LIN {X 46.511,Y 61.150,Z 69.018,A 180.000,B 0.000,C 180.000} C_DIS
LIN {X 46.612,Y 61.449,Z 69.014,A 180.000,B 0.000,C 180.000} C_DIS
LIN {X 46.713,Y 61.747,Z 69.011,A 180.000,B 0.000,C 180.000} C_DIS
LIN {X 46.814,Y 62.046,Z 69.008,A 180.000,B 0.000,C 180.000} C_DIS
LIN {X 46.914,Y 62.344,Z 69.005,A 180.000,B 0.000,C 180.000} C_DIS
LIN {X 47.015,Y 62.643,Z 69.003,A 180.000,B 0.000,C 180.000} C_DIS
LIN {X 47.116,Y 62.941,Z 69.002,A 180.000,B 0.000,C 180.000} C_DIS
LIN {X 47.216,Y 63.240,Z 69.001,A 180.000,B 0.000,C 180.000} C_DIS
LIN {X 47.317,Y 63.538,Z 69.000,A 180.000,B 0.000,C 180.000} C_DIS
LIN {X 47.391,Y 63.759,Z 69.000,A 180.000,B 0.000,C 180.000} C_DIS
; Cutting Move Starts
LIN {X 50.248,Y 72.226,Z 69.000,A 180.000,B 0.000,C 180.000} C_DIS
LIN {X 50.311,Y 72.405,Z 69.000,A 180.000,B 0.000,C 180.000} C_DIS
LIN {X 50.388,Y 72.584,Z 69.000,A 180.000,B 0.000,C 180.000} C_DIS
LIN {X 50.416,Y 72.640,Z 69.000,A 180.000,B 0.000,C 180.000} C_DIS
LIN {X 50.484,Y 72.763,Z 69.000,A 180.000,B 0.000,C 180.000} C_DIS
LIN {X 50.595,Y 72.936,Z 69.000,A 180.000,B 0.000,C 180.000} C_DIS
LIN {X 50.599,Y 72.941,Z 69.000,A 180.000,B 0.000,C 180.000} C_DIS
LIN {X 50.665,Y 73.031,Z 69.000,A 180.000,B 0.000,C 180.000} C_DIS
LIN {X 50.737,Y 73.120,Z 69.000,A 180.000,B 0.000,C 180.000} C_DIS
LIN {X 50.774,Y 73.162,Z 69.000,A 180.000,B 0.000,C 180.000} C_DIS
LIN {X 50.905,Y 73.299,Z 69.000,A 180.000,B 0.000,C 180.000} C_DIS
LIN {X 50.953,Y 73.343,Z 69.000,A 180.000,B 0.000,C 180.000} C_DIS
LIN {X 51.112,Y 73.478,Z 69.000,A 180.000,B 0.000,C 180.000} C_DIS
LIN {X 51.131,Y 73.493,Z 69.000,A 180.000,B 0.000,C 180.000} C_DIS
LIN {X 51.310,Y 73.616,Z 69.000,A 180.000,B 0.000,C 180.000} C_DIS
LIN {X 51.376,Y 73.656,Z 69.000,A 180.000,B 0.000,C 180.000} C_DIS
LIN {X 51.489,Y 73.719,Z 69.000,A 180.000,B 0.000,C 180.000} C_DIS
LIN {X 51.668,Y 73.803,Z 69.000,A 180.000,B 0.000,C 180.000} C_DIS
LIN {X 51.749,Y 73.835,Z 69.000,A 180.000,B 0.000,C 180.000} C_DIS
LIN {X 51.847,Y 73.870,Z 69.000,A 180.000,B 0.000,C 180.000} C_DIS
LIN {X 52.025,Y 73.923,Z 69.000,A 180.000,B 0.000,C 180.000} C_DIS
LIN {X 52.204,Y 73.961,Z 69.000,A 180.000,B 0.000,C 180.000} C_DIS
LIN {X 52.383,Y 73.987,Z 69.000,A 180.000,B 0.000,C 180.000} C_DIS
LIN {X 52.562,Y 73.999,Z 69.000,A 180.000,B 0.000,C 180.000} C_DIS
LIN {X 52.740,Y 73.998,Z 69.000,A 180.000,B 0.000,C 180.000} C_DIS
LIN {X 52.919,Y 73.985,Z 69.000,A 180.000,B 0.000,C 180.000} C_DIS
LIN {X 53.098,Y 73.958,Z 69.000,A 180.000,B 0.000,C 180.000} C_DIS
LIN {X 53.277,Y 73.918,Z 69.000,A 180.000,B 0.000,C 180.000} C_DIS
LIN {X 53.455,Y 73.864,Z 69.000,A 180.000,B 0.000,C 180.000} C_DIS
LIN {X 83.198,Y 63.830,Z 69.000,A 180.000,B 0.000,C 180.000} C_DIS
LIN {X 96.464,Y 59.355,Z 69.000,A 180.000,B 0.000,C 180.000} C_DIS
LIN {X 96.539,Y 59.329,Z 69.000,A 180.000,B 0.000,C 180.000} C_DIS
LIN {X 96.718,Y 59.257,Z 69.000,A 180.000,B 0.000,C 180.000} C_DIS
LIN {X 96.883,Y 59.176,Z 69.000,A 180.000,B 0.000,C 180.000} C_DIS
LIN {X 96.897,Y 59.169,Z 69.000,A 180.000,B 0.000,C 180.000} C_DIS
LIN {X 97.075,Y 59.061,Z 69.000,A 180.000,B 0.000,C 180.000} C_DIS
LIN {X 97.167,Y 58.997,Z 69.000,A 180.000,B 0.000,C 180.000} C_DIS
LIN {X 97.254,Y 58.931,Z 69.000,A 180.000,B 0.000,C 180.000} C_DIS
LIN {X 97.385,Y 58.819,Z 69.000,A 180.000,B 0.000,C 180.000} C_DIS
LIN {X 97.433,Y 58.774,Z 69.000,A 180.000,B 0.000,C 180.000} C_DIS
LIN {X 97.562,Y 58.640,Z 69.000,A 180.000,B 0.000,C 180.000} C_DIS
LIN {X 97.612,Y 58.582,Z 69.000,A 180.000,B 0.000,C 180.000} C_DIS
LIN {X 97.707,Y 58.461,Z 69.000,A 180.000,B 0.000,C 180.000} C_DIS
LIN {X 97.790,Y 58.341,Z 69.000,A 180.000,B 0.000,C 180.000} C_DIS
LIN {X 97.828,Y 58.282,Z 69.000,A 180.000,B 0.000,C 180.000} C_DIS
LIN {X 97.928,Y 58.103,Z 69.000,A 180.000,B 0.000,C 180.000} C_DIS
LIN {X 97.969,Y 58.017,Z 69.000,A 180.000,B 0.000,C 180.000} C_DIS
LIN {X 98.009,Y 57.925,Z 69.000,A 180.000,B 0.000,C 180.000} C_DIS
LIN {X 98.075,Y 57.746,Z 69.000,A 180.000,B 0.000,C 180.000} C_DIS
LIN {X 98.125,Y 57.567,Z 69.000,A 180.000,B 0.000,C 180.000} C_DIS
LIN {X 98.148,Y 57.466,Z 69.000,A 180.000,B 0.000,C 180.000} C_DIS
LIN {X 98.162,Y 57.388,Z 69.000,A 180.000,B 0.000,C 180.000} C_DIS
LIN {X 98.186,Y 57.210,Z 69.000,A 180.000,B 0.000,C 180.000} C_DIS
LIN {X 98.196,Y 57.031,Z 69.000,A 180.000,B 0.000,C 180.000} C_DIS
LIN {X 98.193,Y 56.852,Z 69.000,A 180.000,B 0.000,C 180.000} C_DIS
LIN {X 98.178,Y 56.673,Z 69.000,A 180.000,B 0.000,C 180.000} C_DIS
LIN {X 98.150,Y 56.495,Z 69.000,A 180.000,B 0.000,C 180.000} C_DIS
LIN {X 98.148,Y 56.485,Z 69.000,A 180.000,B 0.000,C 180.000} C_DIS
LIN {X 98.108,Y 56.316,Z 69.000,A 180.000,B 0.000,C 180.000} C_DIS
LIN {X 98.052,Y 56.137,Z 69.000,A 180.000,B 0.000,C 180.000} C_DIS
LIN {X 97.793,Y 55.369,Z 69.000,A 180.000,B 0.000,C 180.000} C_DIS
LIN {X 97.793,Y 55.367,Z 69.000,A 180.000,B 0.000,C 180.000} C_DIS
LIN {X 97.971,Y 55.243,Z 69.000,A 180.000,B 0.000,C 180.000} C_DIS
LIN {X 98.148,Y 55.119,Z 69.000,A 180.000,B 0.000,C 180.000} C_DIS
LIN {X 98.220,Y 55.064,Z 69.000,A 180.000,B 0.000,C 180.000} C_DIS
LIN {X 98.505,Y 54.838,Z 69.000,A 180.000,B 0.000,C 180.000} C_DIS
LIN {X 98.665,Y 54.707,Z 69.000,A 180.000,B 0.000,C 180.000} C_DIS
LIN {X 98.684,Y 54.690,Z 69.000,A 180.000,B 0.000,C 180.000} C_DIS
LIN {X 98.863,Y 54.528,Z 69.000,A 180.000,B 0.000,C 180.000} C_DIS
LIN {X 99.042,Y 54.367,Z 69.000,A 180.000,B 0.000,C 180.000} C_DIS
LIN {X 99.060,Y 54.349,Z 69.000,A 180.000,B 0.000,C 180.000} C_DIS
LIN {X 99.221,Y 54.188,Z 69.000,A 180.000,B 0.000,C 180.000} C_DIS
LIN {X 99.412,Y 53.992,Z 69.000,A 180.000,B 0.000,C 180.000} C_DIS
LIN {X 99.575,Y 53.813,Z 69.000,A 180.000,B 0.000,C 180.000} C_DIS
LIN {X 99.757,Y 53.602,Z 69.000,A 180.000,B 0.000,C 180.000} C_DIS
LIN {X 99.881,Y 53.455,Z 69.000,A 180.000,B 0.000,C 180.000} C_DIS
LIN {X 99.936,Y 53.385,Z 69.000,A 180.000,B 0.000,C 180.000} C_DIS
LIN {X 100.153,Y 53.098,Z 69.000,A 180.000,B 0.000,C 180.000} C_DIS
LIN {X 100.282,Y 52.919,Z 69.000,A 180.000,B 0.000,C 180.000} C_DIS
LIN {X 100.520,Y 52.562,Z 69.000,A 180.000,B 0.000,C 180.000} C_DIS
LIN {X 100.629,Y 52.383,Z 69.000,A 180.000,B 0.000,C 180.000} C_DIS
LIN {X 100.732,Y 52.204,Z 69.000,A 180.000,B 0.000,C 180.000} C_DIS
LIN {X 100.829,Y 52.034,Z 69.000,A 180.000,B 0.000,C 180.000} C_DIS
LIN {X 100.835,Y 52.025,Z 69.000,A 180.000,B 0.000,C 180.000} C_DIS
LIN {X 100.927,Y 51.847,Z 69.000,A 180.000,B 0.000,C 180.000} C_DIS
LIN {X 101.016,Y 51.668,Z 69.000,A 180.000,B 0.000,C 180.000} C_DIS
LIN {X 101.104,Y 51.489,Z 69.000,A 180.000,B 0.000,C 180.000} C_DIS
LIN {X 101.183,Y 51.310,Z 69.000,A 180.000,B 0.000,C 180.000} C_DIS
LIN {X 101.258,Y 51.131,Z 69.000,A 180.000,B 0.000,C 180.000} C_DIS
LIN {X 101.333,Y 50.953,Z 69.000,A 180.000,B 0.000,C 180.000} C_DIS
LIN {X 101.366,Y 50.869,Z 69.000,A 180.000,B 0.000,C 180.000} C_DIS
LIN {X 101.399,Y 50.774,Z 69.000,A 180.000,B 0.000,C 180.000} C_DIS
LIN {X 101.523,Y 50.416,Z 69.000,A 180.000,B 0.000,C 180.000} C_DIS
LIN {X 101.545,Y 50.354,Z 69.000,A 180.000,B 0.000,C 180.000} C_DIS
LIN {X 101.579,Y 50.238,Z 69.000,A 180.000,B 0.000,C 180.000} C_DIS
LIN {X 101.679,Y 49.880,Z 69.000,A 180.000,B 0.000,C 180.000} C_DIS
LIN {X 101.723,Y 49.708,Z 69.000,A 180.000,B 0.000,C 180.000} C_DIS
LIN {X 101.725,Y 49.701,Z 69.000,A 180.000,B 0.000,C 180.000} C_DIS
LIN {X 101.763,Y 49.523,Z 69.000,A 180.000,B 0.000,C 180.000} C_DIS
LIN {X 101.801,Y 49.344,Z 69.000,A 180.000,B 0.000,C 180.000} C_DIS
LIN {X 101.837,Y 49.165,Z 69.000,A 180.000,B 0.000,C 180.000} C_DIS
LIN {X 101.864,Y 48.986,Z 69.000,A 180.000,B 0.000,C 180.000} C_DIS
LIN {X 101.902,Y 48.729,Z 69.000,A 180.000,B 0.000,C 180.000} C_DIS
LIN {X 101.917,Y 48.629,Z 69.000,A 180.000,B 0.000,C 180.000} C_DIS
LIN {X 101.935,Y 48.450,Z 69.000,A 180.000,B 0.000,C 180.000} C_DIS
LIN {X 101.964,Y 48.092,Z 69.000,A 180.000,B 0.000,C 180.000} C_DIS
LIN {X 101.974,Y 47.914,Z 69.000,A 180.000,B 0.000,C 180.000} C_DIS
LIN {X 101.982,Y 47.556,Z 69.000,A 180.000,B 0.000,C 180.000} C_DIS
LIN {X 101.983,Y 47.377,Z 69.000,A 180.000,B 0.000,C 180.000} C_DIS
LIN {X 101.977,Y 47.198,Z 69.000,A 180.000,B 0.000,C 180.000} C_DIS
LIN {X 101.969,Y 47.020,Z 69.000,A 180.000,B 0.000,C 180.000} C_DIS
LIN {X 101.961,Y 46.841,Z 69.000,A 180.000,B 0.000,C 180.000} C_DIS
LIN {X 101.945,Y 46.662,Z 69.000,A 180.000,B 0.000,C 180.000} C_DIS
LIN {X 101.907,Y 46.305,Z 69.000,A 180.000,B 0.000,C 180.000} C_DIS
LIN {X 101.902,Y 46.257,Z 69.000,A 180.000,B 0.000,C 180.000} C_DIS
LIN {X 101.883,Y 46.126,Z 69.000,A 180.000,B 0.000,C 180.000} C_DIS
LIN {X 101.822,Y 45.768,Z 69.000,A 180.000,B 0.000,C 180.000} C_DIS
LIN {X 101.790,Y 45.590,Z 69.000,A 180.000,B 0.000,C 180.000} C_DIS
LIN {X 101.748,Y 45.411,Z 69.000,A 180.000,B 0.000,C 180.000} C_DIS
LIN {X 101.706,Y 45.232,Z 69.000,A 180.000,B 0.000,C 180.000} C_DIS
LIN {X 101.663,Y 45.053,Z 69.000,A 180.000,B 0.000,C 180.000} C_DIS
LIN {X 101.611,Y 44.874,Z 69.000,A 180.000,B 0.000,C 180.000} C_DIS
LIN {X 101.545,Y 44.655,Z 69.000,A 180.000,B 0.000,C 180.000} C_DIS
LIN {X 101.503,Y 44.517,Z 69.000,A 180.000,B 0.000,C 180.000} C_DIS
LIN {X 101.439,Y 44.338,Z 69.000,A 180.000,B 0.000,C 180.000} C_DIS
LIN {X 101.306,Y 43.981,Z 69.000,A 180.000,B 0.000,C 180.000} C_DIS
LIN {X 101.232,Y 43.802,Z 69.000,A 180.000,B 0.000,C 180.000} C_DIS
LIN {X 101.072,Y 43.444,Z 69.000,A 180.000,B 0.000,C 180.000} C_DIS
LIN {X 101.008,Y 43.311,Z 69.000,A 180.000,B 0.000,C 180.000} C_DIS
LIN {X 100.985,Y 43.266,Z 69.000,A 180.000,B 0.000,C 180.000} C_DIS
LIN {X 100.797,Y 42.908,Z 69.000,A 180.000,B 0.000,C 180.000} C_DIS
LIN {X 100.695,Y 42.729,Z 69.000,A 180.000,B 0.000,C 180.000} C_DIS
LIN {X 100.586,Y 42.550,Z 69.000,A 180.000,B 0.000,C 180.000} C_DIS
LIN {X 100.478,Y 42.372,Z 69.000,A 180.000,B 0.000,C 180.000} C_DIS
LIN {X 100.472,Y 42.362,Z 69.000,A 180.000,B 0.000,C 180.000} C_DIS
LIN {X 100.357,Y 42.193,Z 69.000,A 180.000,B 0.000,C 180.000} C_DIS
LIN {X 100.233,Y 42.014,Z 69.000,A 180.000,B 0.000,C 180.000} C_DIS
LIN {X 100.114,Y 41.846,Z 69.000,A 180.000,B 0.000,C 180.000} C_DIS
LIN {X 100.107,Y 41.835,Z 69.000,A 180.000,B 0.000,C 180.000} C_DIS
LIN {X 99.966,Y 41.657,Z 69.000,A 180.000,B 0.000,C 180.000} C_DIS
LIN {X 99.824,Y 41.478,Z 69.000,A 180.000,B 0.000,C 180.000} C_DIS
LIN {X 99.757,Y 41.394,Z 69.000,A 180.000,B 0.000,C 180.000} C_DIS
LIN {X 99.675,Y 41.299,Z 69.000,A 180.000,B 0.000,C 180.000} C_DIS
LIN {X 99.399,Y 40.994,Z 69.000,A 180.000,B 0.000,C 180.000} C_DIS
LIN {X 99.351,Y 40.942,Z 69.000,A 180.000,B 0.000,C 180.000} C_DIS
LIN {X 99.221,Y 40.811,Z 69.000,A 180.000,B 0.000,C 180.000} C_DIS
LIN {X 98.988,Y 40.584,Z 69.000,A 180.000,B 0.000,C 180.000} C_DIS
LIN {X 98.863,Y 40.468,Z 69.000,A 180.000,B 0.000,C 180.000} C_DIS
LIN {X 98.790,Y 40.405,Z 69.000,A 180.000,B 0.000,C 180.000} C_DIS
LIN {X 98.583,Y 40.226,Z 69.000,A 180.000,B 0.000,C 180.000} C_DIS
LIN {X 98.505,Y 40.160,Z 69.000,A 180.000,B 0.000,C 180.000} C_DIS
LIN {X 98.363,Y 40.048,Z 69.000,A 180.000,B 0.000,C 180.000} C_DIS
LIN {X 98.127,Y 39.869,Z 69.000,A 180.000,B 0.000,C 180.000} C_DIS
LIN {X 97.969,Y 39.752,Z 69.000,A 180.000,B 0.000,C 180.000} C_DIS
LIN {X 97.878,Y 39.690,Z 69.000,A 180.000,B 0.000,C 180.000} C_DIS
LIN {X 97.608,Y 39.511,Z 69.000,A 180.000,B 0.000,C 180.000} C_DIS
LIN {X 97.433,Y 39.400,Z 69.000,A 180.000,B 0.000,C 180.000} C_DIS
LIN {X 97.315,Y 39.333,Z 69.000,A 180.000,B 0.000,C 180.000} C_DIS
LIN {X 97.075,Y 39.194,Z 69.000,A 180.000,B 0.000,C 180.000} C_DIS
LIN {X 97.004,Y 39.154,Z 69.000,A 180.000,B 0.000,C 180.000} C_DIS
LIN {X 96.897,Y 39.098,Z 69.000,A 180.000,B 0.000,C 180.000} C_DIS
LIN {X 96.539,Y 38.920,Z 69.000,A 180.000,B 0.000,C 180.000} C_DIS
LIN {X 96.360,Y 38.838,Z 69.000,A 180.000,B 0.000,C 180.000} C_DIS
LIN {X 96.003,Y 38.688,Z 69.000,A 180.000,B 0.000,C 180.000} C_DIS
LIN {X 95.824,Y 38.618,Z 69.000,A 180.000,B 0.000,C 180.000} C_DIS
LIN {X 95.466,Y 38.494,Z 69.000,A 180.000,B 0.000,C 180.000} C_DIS
LIN {X 95.301,Y 38.439,Z 69.000,A 180.000,B 0.000,C 180.000} C_DIS
LIN {X 95.288,Y 38.435,Z 69.000,A 180.000,B 0.000,C 180.000} C_DIS
LIN {X 95.109,Y 38.385,Z 69.000,A 180.000,B 0.000,C 180.000} C_DIS
LIN {X 94.930,Y 38.335,Z 69.000,A 180.000,B 0.000,C 180.000} C_DIS
LIN {X 94.751,Y 38.287,Z 69.000,A 180.000,B 0.000,C 180.000} C_DIS
LIN {X 94.630,Y 38.260,Z 69.000,A 180.000,B 0.000,C 180.000} C_DIS
LIN {X 94.394,Y 38.210,Z 69.000,A 180.000,B 0.000,C 180.000} C_DIS
LIN {X 94.215,Y 38.172,Z 69.000,A 180.000,B 0.000,C 180.000} C_DIS
LIN {X 94.036,Y 38.143,Z 69.000,A 180.000,B 0.000,C 180.000} C_DIS
LIN {X 93.679,Y 38.091,Z 69.000,A 180.000,B 0.000,C 180.000} C_DIS
LIN {X 93.612,Y 38.081,Z 69.000,A 180.000,B 0.000,C 180.000} C_DIS
LIN {X 93.500,Y 38.070,Z 69.000,A 180.000,B 0.000,C 180.000} C_DIS
LIN {X 93.142,Y 38.040,Z 69.000,A 180.000,B 0.000,C 180.000} C_DIS
LIN {X 92.964,Y 38.027,Z 69.000,A 180.000,B 0.000,C 180.000} C_DIS
LIN {X 92.785,Y 38.023,Z 69.000,A 180.000,B 0.000,C 180.000} C_DIS
LIN {X 92.606,Y 38.019,Z 69.000,A 180.000,B 0.000,C 180.000} C_DIS
LIN {X 92.427,Y 38.016,Z 69.000,A 180.000,B 0.000,C 180.000} C_DIS
LIN {X 92.249,Y 38.021,Z 69.000,A 180.000,B 0.000,C 180.000} C_DIS
LIN {X 91.946,Y 38.034,Z 69.000,A 180.000,B 0.000,C 180.000} C_DIS
LIN {X 91.944,Y 38.032,Z 69.000,A 180.000,B 0.000,C 180.000} C_DIS
LIN {X 91.712,Y 37.344,Z 69.000,A 180.000,B 0.000,C 180.000} C_DIS
LIN {X 91.659,Y 37.187,Z 69.000,A 180.000,B 0.000,C 180.000} C_DIS
LIN {X 91.588,Y 37.009,Z 69.000,A 180.000,B 0.000,C 180.000} C_DIS
LIN {X 91.533,Y 36.894,Z 69.000,A 180.000,B 0.000,C 180.000} C_DIS
LIN {X 91.500,Y 36.830,Z 69.000,A 180.000,B 0.000,C 180.000} C_DIS
LIN {X 91.392,Y 36.651,Z 69.000,A 180.000,B 0.000,C 180.000} C_DIS
LIN {X 91.355,Y 36.595,Z 69.000,A 180.000,B 0.000,C 180.000} C_DIS
LIN {X 91.263,Y 36.472,Z 69.000,A 180.000,B 0.000,C 180.000} C_DIS
LIN {X 91.176,Y 36.368,Z 69.000,A 180.000,B 0.000,C 180.000} C_DIS
LIN {X 91.107,Y 36.294,Z 69.000,A 180.000,B 0.000,C 180.000} C_DIS
LIN {X 90.997,Y 36.186,Z 69.000,A 180.000,B 0.000,C 180.000} C_DIS
LIN {X 90.917,Y 36.115,Z 69.000,A 180.000,B 0.000,C 180.000} C_DIS
LIN {X 90.818,Y 36.036,Z 69.000,A 180.000,B 0.000,C 180.000} C_DIS
LIN {X 90.677,Y 35.936,Z 69.000,A 180.000,B 0.000,C 180.000} C_DIS
LIN {X 90.640,Y 35.912,Z 69.000,A 180.000,B 0.000,C 180.000} C_DIS
LIN {X 90.461,Y 35.809,Z 69.000,A 180.000,B 0.000,C 180.000} C_DIS
LIN {X 90.356,Y 35.757,Z 69.000,A 180.000,B 0.000,C 180.000} C_DIS
LIN {X 90.282,Y 35.724,Z 69.000,A 180.000,B 0.000,C 180.000} C_DIS
LIN {X 90.103,Y 35.656,Z 69.000,A 180.000,B 0.000,C 180.000} C_DIS
LIN {X 89.925,Y 35.603,Z 69.000,A 180.000,B 0.000,C 180.000} C_DIS
LIN {X 89.819,Y 35.578,Z 69.000,A 180.000,B 0.000,C 180.000} C_DIS
LIN {X 89.746,Y 35.564,Z 69.000,A 180.000,B 0.000,C 180.000} C_DIS
LIN {X 89.567,Y 35.539,Z 69.000,A 180.000,B 0.000,C 180.000} C_DIS
LIN {X 89.388,Y 35.526,Z 69.000,A 180.000,B 0.000,C 180.000} C_DIS
LIN {X 89.209,Y 35.526,Z 69.000,A 180.000,B 0.000,C 180.000} C_DIS
LIN {X 89.031,Y 35.540,Z 69.000,A 180.000,B 0.000,C 180.000} C_DIS
LIN {X 88.852,Y 35.566,Z 69.000,A 180.000,B 0.000,C 180.000} C_DIS
LIN {X 88.788,Y 35.578,Z 69.000,A 180.000,B 0.000,C 180.000} C_DIS
LIN {X 88.673,Y 35.605,Z 69.000,A 180.000,B 0.000,C 180.000} C_DIS
LIN {X 88.494,Y 35.659,Z 69.000,A 180.000,B 0.000,C 180.000} C_DIS
LIN {X 66.460,Y 43.092,Z 69.000,A 180.000,B 0.000,C 180.000} C_DIS
LIN {X 45.590,Y 50.133,Z 69.000,A 180.000,B 0.000,C 180.000} C_DIS
LIN {X 45.411,Y 50.194,Z 69.000,A 180.000,B 0.000,C 180.000} C_DIS
LIN {X 45.296,Y 50.238,Z 69.000,A 180.000,B 0.000,C 180.000} C_DIS
LIN {X 45.232,Y 50.265,Z 69.000,A 180.000,B 0.000,C 180.000} C_DIS
LIN {X 45.053,Y 50.353,Z 69.000,A 180.000,B 0.000,C 180.000} C_DIS
LIN {X 44.944,Y 50.416,Z 69.000,A 180.000,B 0.000,C 180.000} C_DIS
LIN {X 44.874,Y 50.461,Z 69.000,A 180.000,B 0.000,C 180.000} C_DIS
LIN {X 44.785,Y 50.522,Z 69.000,A 180.000,B 0.000,C 180.000} C_DIS
LIN {X 44.696,Y 50.590,Z 69.000,A 180.000,B 0.000,C 180.000} C_DIS
LIN {X 44.689,Y 50.595,Z 69.000,A 180.000,B 0.000,C 180.000} C_DIS
LIN {X 44.603,Y 50.667,Z 69.000,A 180.000,B 0.000,C 180.000} C_DIS
LIN {X 44.517,Y 50.746,Z 69.000,A 180.000,B 0.000,C 180.000} C_DIS
LIN {X 44.488,Y 50.774,Z 69.000,A 180.000,B 0.000,C 180.000} C_DIS
LIN {X 44.410,Y 50.855,Z 69.000,A 180.000,B 0.000,C 180.000} C_DIS
LIN {X 44.338,Y 50.936,Z 69.000,A 180.000,B 0.000,C 180.000} C_DIS
LIN {X 44.325,Y 50.953,Z 69.000,A 180.000,B 0.000,C 180.000} C_DIS
LIN {X 44.254,Y 51.042,Z 69.000,A 180.000,B 0.000,C 180.000} C_DIS
LIN {X 44.189,Y 51.131,Z 69.000,A 180.000,B 0.000,C 180.000} C_DIS
LIN {X 44.159,Y 51.176,Z 69.000,A 180.000,B 0.000,C 180.000} C_DIS
LIN {X 44.077,Y 51.310,Z 69.000,A 180.000,B 0.000,C 180.000} C_DIS
LIN {X 43.984,Y 51.489,Z 69.000,A 180.000,B 0.000,C 180.000} C_DIS
LIN {X 43.981,Y 51.497,Z 69.000,A 180.000,B 0.000,C 180.000} C_DIS
LIN {X 43.909,Y 51.668,Z 69.000,A 180.000,B 0.000,C 180.000} C_DIS
LIN {X 43.849,Y 51.847,Z 69.000,A 180.000,B 0.000,C 180.000} C_DIS
LIN {X 43.804,Y 52.025,Z 69.000,A 180.000,B 0.000,C 180.000} C_DIS
LIN {X 43.802,Y 52.035,Z 69.000,A 180.000,B 0.000,C 180.000} C_DIS
LIN {X 43.772,Y 52.204,Z 69.000,A 180.000,B 0.000,C 180.000} C_DIS
LIN {X 43.754,Y 52.383,Z 69.000,A 180.000,B 0.000,C 180.000} C_DIS
LIN {X 43.748,Y 52.562,Z 69.000,A 180.000,B 0.000,C 180.000} C_DIS
LIN {X 43.756,Y 52.740,Z 69.000,A 180.000,B 0.000,C 180.000} C_DIS
LIN {X 43.776,Y 52.919,Z 69.000,A 180.000,B 0.000,C 180.000} C_DIS
LIN {X 43.802,Y 53.064,Z 69.000,A 180.000,B 0.000,C 180.000} C_DIS
LIN {X 43.809,Y 53.098,Z 69.000,A 180.000,B 0.000,C 180.000} C_DIS
LIN {X 43.856,Y 53.277,Z 69.000,A 180.000,B 0.000,C 180.000} C_DIS
LIN {X 43.916,Y 53.455,Z 69.000,A 180.000,B 0.000,C 180.000} C_DIS
LIN {X 47.391,Y 63.759,Z 69.000,A 180.000,B 0.000,C 180.000} C_DIS
; Link Move Starts
LIN {X 47.492,Y 64.057,Z 69.000,A 180.000,B 0.000,C 180.000} C_DIS
LIN {X 47.593,Y 64.356,Z 68.999,A 180.000,B 0.000,C 180.000} C_DIS
LIN {X 47.693,Y 64.654,Z 68.998,A 180.000,B 0.000,C 180.000} C_DIS
LIN {X 47.794,Y 64.953,Z 68.996,A 180.000,B 0.000,C 180.000} C_DIS
LIN {X 47.895,Y 65.251,Z 68.994,A 180.000,B 0.000,C 180.000} C_DIS
LIN {X 47.996,Y 65.550,Z 68.991,A 180.000,B 0.000,C 180.000} C_DIS
LIN {X 48.096,Y 65.848,Z 68.988,A 180.000,B 0.000,C 180.000} C_DIS
LIN {X 48.197,Y 66.147,Z 68.985,A 180.000,B 0.000,C 180.000} C_DIS
LIN {X 48.298,Y 66.445,Z 68.981,A 180.000,B 0.000,C 180.000} C_DIS
LIN {X 48.398,Y 66.743,Z 68.977,A 180.000,B 0.000,C 180.000} C_DIS
LIN {X 48.499,Y 67.042,Z 68.972,A 180.000,B 0.000,C 180.000} C_DIS
LIN {X 48.549,Y 67.191,Z 68.969,A 180.000,B 0.000,C 180.000} C_DIS
LIN {X 48.600,Y 67.340,Z 68.967,A 180.000,B 0.000,C 180.000} C_DIS
LIN {X 48.650,Y 67.490,Z 68.964,A 180.000,B 0.000,C 180.000} C_DIS
LIN {X 48.700,Y 67.639,Z 68.961,A 180.000,B 0.000,C 180.000} C_DIS
LIN {X 48.751,Y 67.788,Z 68.959,A 180.000,B 0.000,C 180.000} C_DIS
LIN {X 48.801,Y 67.937,Z 68.956,A 180.000,B 0.000,C 180.000} C_DIS
LIN {X 48.851,Y 68.087,Z 68.952,A 180.000,B 0.000,C 180.000} C_DIS
LIN {X 48.902,Y 68.236,Z 68.949,A 180.000,B 0.000,C 180.000} C_DIS
LIN {X 48.952,Y 68.385,Z 68.946,A 180.000,B 0.000,C 180.000} C_DIS
LIN {X 49.002,Y 68.534,Z 68.943,A 180.000,B 0.000,C 180.000} C_DIS
LIN {X 49.053,Y 68.684,Z 68.939,A 180.000,B 0.000,C 180.000} C_DIS
LIN {X 49.103,Y 68.833,Z 68.936,A 180.000,B 0.000,C 180.000} C_DIS
LIN {X 49.153,Y 68.982,Z 68.932,A 180.000,B 0.000,C 180.000} C_DIS
LIN {X 49.204,Y 69.131,Z 68.928,A 180.000,B 0.000,C 180.000} C_DIS
LIN {X 49.254,Y 69.280,Z 68.925,A 180.000,B 0.000,C 180.000} C_DIS
LIN {X 49.304,Y 69.430,Z 68.921,A 180.000,B 0.000,C 180.000} C_DIS
LIN {X 49.355,Y 69.579,Z 68.917,A 180.000,B 0.000,C 180.000} C_DIS
LIN {X 49.405,Y 69.728,Z 68.913,A 180.000,B 0.000,C 180.000} C_DIS
LIN {X 49.456,Y 69.877,Z 68.909,A 180.000,B 0.000,C 180.000} C_DIS
LIN {X 49.506,Y 70.027,Z 68.905,A 180.000,B 0.000,C 180.000} C_DIS
LIN {X 49.556,Y 70.176,Z 68.900,A 180.000,B 0.000,C 180.000} C_DIS
LIN {X 49.607,Y 70.325,Z 68.896,A 180.000,B 0.000,C 180.000} C_DIS
LIN {X 49.657,Y 70.474,Z 68.892,A 180.000,B 0.000,C 180.000} C_DIS
LIN {X 49.707,Y 70.624,Z 68.887,A 180.000,B 0.000,C 180.000} C_DIS
LIN {X 49.758,Y 70.773,Z 68.883,A 180.000,B 0.000,C 180.000} C_DIS
LIN {X 49.808,Y 70.922,Z 68.878,A 180.000,B 0.000,C 180.000} C_DIS
LIN {X 49.858,Y 71.071,Z 68.873,A 180.000,B 0.000,C 180.000} C_DIS
LIN {X 49.909,Y 71.221,Z 68.869,A 180.000,B 0.000,C 180.000} C_DIS
LIN {X 49.959,Y 71.370,Z 68.864,A 180.000,B 0.000,C 180.000} C_DIS
LIN {X 50.009,Y 71.519,Z 68.859,A 180.000,B 0.000,C 180.000} C_DIS
LIN {X 50.060,Y 71.668,Z 68.854,A 180.000,B 0.000,C 180.000} C_DIS
LIN {X 50.085,Y 71.743,Z 68.851,A 180.000,B 0.000,C 180.000} C_DIS
LIN {X 50.110,Y 71.818,Z 68.849,A 180.000,B 0.000,C 180.000} C_DIS
LIN {X 50.135,Y 71.892,Z 68.846,A 180.000,B 0.000,C 180.000} C_DIS
LIN {X 50.160,Y 71.967,Z 68.844,A 180.000,B 0.000,C 180.000} C_DIS
LIN {X 50.186,Y 72.041,Z 68.841,A 180.000,B 0.000,C 180.000} C_DIS
LIN {X 50.211,Y 72.116,Z 68.839,A 180.000,B 0.000,C 180.000} C_DIS
LIN {X 50.236,Y 72.191,Z 68.836,A 180.000,B 0.000,C 180.000} C_DIS
LIN {X 50.261,Y 72.265,Z 68.833,A 180.000,B 0.000,C 180.000} C_DIS
LIN {X 50.287,Y 72.340,Z 68.831,A 180.000,B 0.000,C 180.000} C_DIS
LIN {X 50.314,Y 72.413,Z 68.828,A 180.000,B 0.000,C 180.000} C_DIS
LIN {X 50.344,Y 72.486,Z 68.825,A 180.000,B 0.000,C 180.000} C_DIS
LIN {X 50.376,Y 72.558,Z 68.823,A 180.000,B 0.000,C 180.000} C_DIS
LIN {X 50.411,Y 72.629,Z 68.820,A 180.000,B 0.000,C 180.000} C_DIS
LIN {X 50.447,Y 72.699,Z 68.817,A 180.000,B 0.000,C 180.000} C_DIS
LIN {X 50.486,Y 72.767,Z 68.815,A 180.000,B 0.000,C 180.000} C_DIS
LIN {X 50.527,Y 72.835,Z 68.812,A 180.000,B 0.000,C 180.000} C_DIS
LIN {X 50.570,Y 72.900,Z 68.809,A 180.000,B 0.000,C 180.000} C_DIS
LIN {X 50.616,Y 72.965,Z 68.807,A 180.000,B 0.000,C 180.000} C_DIS
LIN {X 50.663,Y 73.028,Z 68.804,A 180.000,B 0.000,C 180.000} C_DIS
LIN {X 50.712,Y 73.090,Z 68.801,A 180.000,B 0.000,C 180.000} C_DIS
LIN {X 50.763,Y 73.150,Z 68.798,A 180.000,B 0.000,C 180.000} C_DIS
LIN {X 50.816,Y 73.208,Z 68.796,A 180.000,B 0.000,C 180.000} C_DIS
LIN {X 50.870,Y 73.265,Z 68.793,A 180.000,B 0.000,C 180.000} C_DIS
LIN {X 50.927,Y 73.320,Z 68.790,A 180.000,B 0.000,C 180.000} C_DIS
LIN {X 50.985,Y 73.373,Z 68.787,A 180.000,B 0.000,C 180.000} C_DIS
LIN {X 51.045,Y 73.424,Z 68.785,A 180.000,B 0.000,C 180.000} C_DIS
LIN {X 51.106,Y 73.473,Z 68.782,A 180.000,B 0.000,C 180.000} C_DIS
LIN {X 51.169,Y 73.521,Z 68.779,A 180.000,B 0.000,C 180.000} C_DIS
LIN {X 51.234,Y 73.566,Z 68.776,A 180.000,B 0.000,C 180.000} C_DIS
LIN {X 51.299,Y 73.609,Z 68.774,A 180.000,B 0.000,C 180.000} C_DIS
LIN {X 51.366,Y 73.651,Z 68.771,A 180.000,B 0.000,C 180.000} C_DIS
LIN {X 51.435,Y 73.690,Z 68.768,A 180.000,B 0.000,C 180.000} C_DIS
LIN {X 51.504,Y 73.727,Z 68.765,A 180.000,B 0.000,C 180.000} C_DIS
LIN {X 51.575,Y 73.761,Z 68.763,A 180.000,B 0.000,C 180.000} C_DIS
LIN {X 51.647,Y 73.794,Z 68.760,A 180.000,B 0.000,C 180.000} C_DIS
LIN {X 51.720,Y 73.824,Z 68.757,A 180.000,B 0.000,C 180.000} C_DIS
LIN {X 51.793,Y 73.852,Z 68.754,A 180.000,B 0.000,C 180.000} C_DIS
LIN {X 51.868,Y 73.877,Z 68.752,A 180.000,B 0.000,C 180.000} C_DIS
LIN {X 51.943,Y 73.901,Z 68.749,A 180.000,B 0.000,C 180.000} C_DIS
LIN {X 52.019,Y 73.921,Z 68.746,A 180.000,B 0.000,C 180.000} C_DIS
LIN {X 52.096,Y 73.940,Z 68.743,A 180.000,B 0.000,C 180.000} C_DIS
LIN {X 52.173,Y 73.956,Z 68.741,A 180.000,B 0.000,C 180.000} C_DIS
LIN {X 52.250,Y 73.969,Z 68.738,A 180.000,B 0.000,C 180.000} C_DIS
LIN {X 52.328,Y 73.980,Z 68.735,A 180.000,B 0.000,C 180.000} C_DIS
LIN {X 52.407,Y 73.989,Z 68.732,A 180.000,B 0.000,C 180.000} C_DIS
LIN {X 52.485,Y 73.995,Z 68.730,A 180.000,B 0.000,C 180.000} C_DIS
LIN {X 52.564,Y 73.999,Z 68.727,A 180.000,B 0.000,C 180.000} C_DIS
LIN {X 52.643,Y 74.000,Z 68.724,A 180.000,B 0.000,C 180.000} C_DIS
LIN {X 52.721,Y 73.999,Z 68.721,A 180.000,B 0.000,C 180.000} C_DIS
LIN {X 52.800,Y 73.995,Z 68.719,A 180.000,B 0.000,C 180.000} C_DIS
LIN {X 52.878,Y 73.989,Z 68.716,A 180.000,B 0.000,C 180.000} C_DIS
LIN {X 52.957,Y 73.980,Z 68.713,A 180.000,B 0.000,C 180.000} C_DIS
LIN {X 53.035,Y 73.969,Z 68.710,A 180.000,B 0.000,C 180.000} C_DIS
LIN {X 53.112,Y 73.955,Z 68.708,A 180.000,B 0.000,C 180.000} C_DIS
LIN {X 53.189,Y 73.939,Z 68.705,A 180.000,B 0.000,C 180.000} C_DIS
LIN {X 53.266,Y 73.921,Z 68.702,A 180.000,B 0.000,C 180.000} C_DIS
LIN {X 53.342,Y 73.900,Z 68.699,A 180.000,B 0.000,C 180.000} C_DIS
LIN {X 53.417,Y 73.877,Z 68.697,A 180.000,B 0.000,C 180.000} C_DIS
LIN {X 53.492,Y 73.852,Z 68.694,A 180.000,B 0.000,C 180.000} C_DIS
LIN {X 53.641,Y 73.801,Z 68.688,A 180.000,B 0.000,C 180.000} C_DIS
LIN {X 53.716,Y 73.776,Z 68.686,A 180.000,B 0.000,C 180.000} C_DIS
LIN {X 53.865,Y 73.726,Z 68.680,A 180.000,B 0.000,C 180.000} C_DIS
LIN {X 54.313,Y 73.575,Z 68.664,A 180.000,B 0.000,C 180.000} C_DIS
LIN {X 54.536,Y 73.499,Z 68.655,A 180.000,B 0.000,C 180.000} C_DIS
LIN {X 54.686,Y 73.449,Z 68.650,A 180.000,B 0.000,C 180.000} C_DIS
LIN {X 55.133,Y 73.298,Z 68.633,A 180.000,B 0.000,C 180.000} C_DIS
LIN {X 55.283,Y 73.247,Z 68.628,A 180.000,B 0.000,C 180.000} C_DIS
LIN {X 55.730,Y 73.096,Z 68.611,A 180.000,B 0.000,C 180.000} C_DIS
LIN {X 55.880,Y 73.046,Z 68.606,A 180.000,B 0.000,C 180.000} C_DIS
LIN {X 56.551,Y 72.819,Z 68.581,A 180.000,B 0.000,C 180.000} C_DIS
LIN {X 57.596,Y 72.467,Z 68.543,A 180.000,B 0.000,C 180.000} C_DIS
LIN {X 58.342,Y 72.215,Z 68.515,A 180.000,B 0.000,C 180.000} C_DIS
LIN {X 61.401,Y 71.183,Z 68.402,A 180.000,B 0.000,C 180.000} C_DIS
LIN {X 61.625,Y 71.108,Z 68.394,A 180.000,B 0.000,C 180.000} C_DIS
LIN {X 62.371,Y 70.856,Z 68.367,A 180.000,B 0.000,C 180.000} C_DIS
LIN {X 62.595,Y 70.780,Z 68.358,A 180.000,B 0.000,C 180.000} C_DIS
LIN {X 62.744,Y 70.730,Z 68.353,A 180.000,B 0.000,C 180.000} C_DIS
LIN {X 63.192,Y 70.579,Z 68.336,A 180.000,B 0.000,C 180.000} C_DIS
LIN {X 63.267,Y 70.554,Z 68.334,A 180.000,B 0.000,C 180.000} C_DIS
LIN {X 63.416,Y 70.504,Z 68.328,A 180.000,B 0.000,C 180.000} C_DIS
LIN {X 63.864,Y 70.353,Z 68.312,A 180.000,B 0.000,C 180.000} C_DIS
LIN {X 64.013,Y 70.302,Z 68.306,A 180.000,B 0.000,C 180.000} C_DIS
LIN {X 64.461,Y 70.151,Z 68.290,A 180.000,B 0.000,C 180.000} C_DIS
LIN {X 64.610,Y 70.101,Z 68.284,A 180.000,B 0.000,C 180.000} C_DIS
LIN {X 64.834,Y 70.025,Z 68.276,A 180.000,B 0.000,C 180.000} C_DIS
LIN {X 64.983,Y 69.975,Z 68.270,A 180.000,B 0.000,C 180.000} C_DIS
LIN {X 65.058,Y 69.950,Z 68.268,A 180.000,B 0.000,C 180.000} C_DIS
LIN {X 65.207,Y 69.899,Z 68.262,A 180.000,B 0.000,C 180.000} C_DIS
LIN {X 65.431,Y 69.824,Z 68.254,A 180.000,B 0.000,C 180.000} C_DIS
LIN {X 65.580,Y 69.774,Z 68.248,A 180.000,B 0.000,C 180.000} C_DIS
LIN {X 65.655,Y 69.748,Z 68.246,A 180.000,B 0.000,C 180.000} C_DIS
LIN {X 65.804,Y 69.698,Z 68.240,A 180.000,B 0.000,C 180.000} C_DIS
LIN {X 66.028,Y 69.623,Z 68.232,A 180.000,B 0.000,C 180.000} C_DIS
LIN {X 66.177,Y 69.572,Z 68.226,A 180.000,B 0.000,C 180.000} C_DIS
LIN {X 66.252,Y 69.547,Z 68.224,A 180.000,B 0.000,C 180.000} C_DIS
LIN {X 66.401,Y 69.497,Z 68.218,A 180.000,B 0.000,C 180.000} C_DIS
LIN {X 66.625,Y 69.421,Z 68.210,A 180.000,B 0.000,C 180.000} C_DIS
LIN {X 66.774,Y 69.371,Z 68.204,A 180.000,B 0.000,C 180.000} C_DIS
LIN {X 66.848,Y 69.346,Z 68.202,A 180.000,B 0.000,C 180.000} C_DIS
LIN {X 66.998,Y 69.295,Z 68.196,A 180.000,B 0.000,C 180.000} C_DIS
LIN {X 67.147,Y 69.245,Z 68.191,A 180.000,B 0.000,C 180.000} C_DIS
LIN {X 67.296,Y 69.195,Z 68.185,A 180.000,B 0.000,C 180.000} C_DIS
LIN {X 67.445,Y 69.144,Z 68.180,A 180.000,B 0.000,C 180.000} C_DIS
LIN {X 67.595,Y 69.094,Z 68.174,A 180.000,B 0.000,C 180.000} C_DIS
LIN {X 67.744,Y 69.044,Z 68.169,A 180.000,B 0.000,C 180.000} C_DIS
LIN {X 67.893,Y 68.993,Z 68.164,A 180.000,B 0.000,C 180.000} C_DIS
LIN {X 67.968,Y 68.968,Z 68.161,A 180.000,B 0.000,C 180.000} C_DIS
LIN {X 68.042,Y 68.943,Z 68.159,A 180.000,B 0.000,C 180.000} C_DIS
LIN {X 68.117,Y 68.918,Z 68.156,A 180.000,B 0.000,C 180.000} C_DIS
LIN {X 68.192,Y 68.893,Z 68.154,A 180.000,B 0.000,C 180.000} C_DIS
LIN {X 68.266,Y 68.867,Z 68.151,A 180.000,B 0.000,C 180.000} C_DIS
LIN {X 68.341,Y 68.842,Z 68.149,A 180.000,B 0.000,C 180.000} C_DIS
LIN {X 68.490,Y 68.792,Z 68.144,A 180.000,B 0.000,C 180.000} C_DIS
LIN {X 68.639,Y 68.742,Z 68.139,A 180.000,B 0.000,C 180.000} C_DIS
LIN {X 68.789,Y 68.691,Z 68.134,A 180.000,B 0.000,C 180.000} C_DIS
LIN {X 68.938,Y 68.641,Z 68.129,A 180.000,B 0.000,C 180.000} C_DIS
LIN {X 69.087,Y 68.590,Z 68.124,A 180.000,B 0.000,C 180.000} C_DIS
LIN {X 69.236,Y 68.540,Z 68.120,A 180.000,B 0.000,C 180.000} C_DIS
LIN {X 69.385,Y 68.490,Z 68.115,A 180.000,B 0.000,C 180.000} C_DIS
LIN {X 69.535,Y 68.439,Z 68.111,A 180.000,B 0.000,C 180.000} C_DIS
LIN {X 69.684,Y 68.389,Z 68.106,A 180.000,B 0.000,C 180.000} C_DIS
LIN {X 69.833,Y 68.339,Z 68.102,A 180.000,B 0.000,C 180.000} C_DIS
LIN {X 69.982,Y 68.288,Z 68.097,A 180.000,B 0.000,C 180.000} C_DIS
LIN {X 70.132,Y 68.238,Z 68.093,A 180.000,B 0.000,C 180.000} C_DIS
LIN {X 70.281,Y 68.188,Z 68.089,A 180.000,B 0.000,C 180.000} C_DIS
LIN {X 70.430,Y 68.137,Z 68.085,A 180.000,B 0.000,C 180.000} C_DIS
LIN {X 70.579,Y 68.087,Z 68.081,A 180.000,B 0.000,C 180.000} C_DIS
LIN {X 70.729,Y 68.037,Z 68.077,A 180.000,B 0.000,C 180.000} C_DIS
LIN {X 70.878,Y 67.986,Z 68.073,A 180.000,B 0.000,C 180.000} C_DIS
LIN {X 71.027,Y 67.936,Z 68.070,A 180.000,B 0.000,C 180.000} C_DIS
LIN {X 71.176,Y 67.886,Z 68.066,A 180.000,B 0.000,C 180.000} C_DIS
LIN {X 71.326,Y 67.835,Z 68.062,A 180.000,B 0.000,C 180.000} C_DIS
LIN {X 71.475,Y 67.785,Z 68.059,A 180.000,B 0.000,C 180.000} C_DIS
LIN {X 71.624,Y 67.735,Z 68.056,A 180.000,B 0.000,C 180.000} C_DIS
LIN {X 71.773,Y 67.684,Z 68.052,A 180.000,B 0.000,C 180.000} C_DIS
LIN {X 71.923,Y 67.634,Z 68.049,A 180.000,B 0.000,C 180.000} C_DIS
LIN {X 72.072,Y 67.584,Z 68.046,A 180.000,B 0.000,C 180.000} C_DIS
LIN {X 72.221,Y 67.533,Z 68.043,A 180.000,B 0.000,C 180.000} C_DIS
LIN {X 72.370,Y 67.483,Z 68.040,A 180.000,B 0.000,C 180.000} C_DIS
LIN {X 72.519,Y 67.433,Z 68.037,A 180.000,B 0.000,C 180.000} C_DIS
LIN {X 72.669,Y 67.382,Z 68.034,A 180.000,B 0.000,C 180.000} C_DIS
LIN {X 72.818,Y 67.332,Z 68.032,A 180.000,B 0.000,C 180.000} C_DIS
LIN {X 72.967,Y 67.282,Z 68.029,A 180.000,B 0.000,C 180.000} C_DIS
LIN {X 73.116,Y 67.231,Z 68.027,A 180.000,B 0.000,C 180.000} C_DIS
LIN {X 73.415,Y 67.130,Z 68.022,A 180.000,B 0.000,C 180.000} C_DIS
LIN {X 73.713,Y 67.030,Z 68.018,A 180.000,B 0.000,C 180.000} C_DIS
LIN {X 74.012,Y 66.929,Z 68.014,A 180.000,B 0.000,C 180.000} C_DIS
LIN {X 74.310,Y 66.828,Z 68.011,A 180.000,B 0.000,C 180.000} C_DIS
LIN {X 74.609,Y 66.728,Z 68.008,A 180.000,B 0.000,C 180.000} C_DIS
LIN {X 74.907,Y 66.627,Z 68.005,A 180.000,B 0.000,C 180.000} C_DIS
LIN {X 75.206,Y 66.526,Z 68.003,A 180.000,B 0.000,C 180.000} C_DIS
LIN {X 75.504,Y 66.426,Z 68.002,A 180.000,B 0.000,C 180.000} C_DIS
LIN {X 75.803,Y 66.325,Z 68.001,A 180.000,B 0.000,C 180.000} C_DIS
LIN {X 76.101,Y 66.224,Z 68.000,A 180.000,B 0.000,C 180.000} C_DIS
LIN {X 76.321,Y 66.150,Z 68.000,A 180.000,B 0.000,C 180.000} C_DIS
; Cutting Move Starts
LIN {X 96.464,Y 59.355,Z 68.000,A 180.000,B 0.000,C 180.000} C_DIS
LIN {X 96.539,Y 59.329,Z 68.000,A 180.000,B 0.000,C 180.000} C_DIS
LIN {X 96.718,Y 59.257,Z 68.000,A 180.000,B 0.000,C 180.000} C_DIS
LIN {X 96.883,Y 59.176,Z 68.000,A 180.000,B 0.000,C 180.000} C_DIS
LIN {X 96.897,Y 59.169,Z 68.000,A 180.000,B 0.000,C 180.000} C_DIS
LIN {X 97.075,Y 59.061,Z 68.000,A 180.000,B 0.000,C 180.000} C_DIS
LIN {X 97.167,Y 58.997,Z 68.000,A 180.000,B 0.000,C 180.000} C_DIS
LIN {X 97.254,Y 58.931,Z 68.000,A 180.000,B 0.000,C 180.000} C_DIS
LIN {X 97.385,Y 58.819,Z 68.000,A 180.000,B 0.000,C 180.000} C_DIS
LIN {X 97.433,Y 58.774,Z 68.000,A 180.000,B 0.000,C 180.000} C_DIS
LIN {X 97.562,Y 58.640,Z 68.000,A 180.000,B 0.000,C 180.000} C_DIS
LIN {X 97.612,Y 58.582,Z 68.000,A 180.000,B 0.000,C 180.000} C_DIS
LIN {X 97.707,Y 58.461,Z 68.000,A 180.000,B 0.000,C 180.000} C_DIS
LIN {X 97.790,Y 58.341,Z 68.000,A 180.000,B 0.000,C 180.000} C_DIS
LIN {X 97.828,Y 58.282,Z 68.000,A 180.000,B 0.000,C 180.000} C_DIS
LIN {X 97.928,Y 58.103,Z 68.000,A 180.000,B 0.000,C 180.000} C_DIS
LIN {X 97.969,Y 58.017,Z 68.000,A 180.000,B 0.000,C 180.000} C_DIS
LIN {X 98.009,Y 57.925,Z 68.000,A 180.000,B 0.000,C 180.000} C_DIS
LIN {X 98.075,Y 57.746,Z 68.000,A 180.000,B 0.000,C 180.000} C_DIS
LIN {X 98.125,Y 57.567,Z 68.000,A 180.000,B 0.000,C 180.000} C_DIS
LIN {X 98.148,Y 57.466,Z 68.000,A 180.000,B 0.000,C 180.000} C_DIS
LIN {X 98.162,Y 57.388,Z 68.000,A 180.000,B 0.000,C 180.000} C_DIS
LIN {X 98.186,Y 57.210,Z 68.000,A 180.000,B 0.000,C 180.000} C_DIS
LIN {X 98.196,Y 57.031,Z 68.000,A 180.000,B 0.000,C 180.000} C_DIS
LIN {X 98.193,Y 56.852,Z 68.000,A 180.000,B 0.000,C 180.000} C_DIS
LIN {X 98.178,Y 56.673,Z 68.000,A 180.000,B 0.000,C 180.000} C_DIS
LIN {X 98.166,Y 56.584,Z 68.000,A 180.000,B 0.000,C 180.000} C_DIS
LIN {X 98.158,Y 56.539,Z 68.000,A 180.000,B 0.000,C 180.000} C_DIS
LIN {X 98.154,Y 56.517,Z 68.000,A 180.000,B 0.000,C 180.000} C_DIS
LIN {X 98.153,Y 56.508,Z 68.000,A 180.000,B 0.000,C 180.000} C_DIS
LIN {X 98.153,Y 56.507,Z 68.000,A 180.000,B 0.000,C 180.000} C_DIS
LIN {X 98.174,Y 56.495,Z 68.000,A 180.000,B 0.000,C 180.000} C_DIS
LIN {X 98.327,Y 56.399,Z 68.000,A 180.000,B 0.000,C 180.000} C_DIS
LIN {X 98.447,Y 56.316,Z 68.000,A 180.000,B 0.000,C 180.000} C_DIS
LIN {X 98.704,Y 56.137,Z 68.000,A 180.000,B 0.000,C 180.000} C_DIS
LIN {X 98.863,Y 56.024,Z 68.000,A 180.000,B 0.000,C 180.000} C_DIS
LIN {X 98.947,Y 55.958,Z 68.000,A 180.000,B 0.000,C 180.000} C_DIS
LIN {X 99.221,Y 55.741,Z 68.000,A 180.000,B 0.000,C 180.000} C_DIS
LIN {X 99.393,Y 55.601,Z 68.000,A 180.000,B 0.000,C 180.000} C_DIS
LIN {X 99.399,Y 55.596,Z 68.000,A 180.000,B 0.000,C 180.000} C_DIS
LIN {X 99.578,Y 55.435,Z 68.000,A 180.000,B 0.000,C 180.000} C_DIS
LIN {X 99.791,Y 55.243,Z 68.000,A 180.000,B 0.000,C 180.000} C_DIS
LIN {X 99.936,Y 55.104,Z 68.000,A 180.000,B 0.000,C 180.000} C_DIS
LIN {X 100.150,Y 54.886,Z 68.000,A 180.000,B 0.000,C 180.000} C_DIS
LIN {X 100.293,Y 54.739,Z 68.000,A 180.000,B 0.000,C 180.000} C_DIS
LIN {X 100.323,Y 54.707,Z 68.000,A 180.000,B 0.000,C 180.000} C_DIS
LIN {X 100.472,Y 54.537,Z 68.000,A 180.000,B 0.000,C 180.000} C_DIS
LIN {X 100.651,Y 54.330,Z 68.000,A 180.000,B 0.000,C 180.000} C_DIS
LIN {X 100.785,Y 54.171,Z 68.000,A 180.000,B 0.000,C 180.000} C_DIS
LIN {X 100.829,Y 54.113,Z 68.000,A 180.000,B 0.000,C 180.000} C_DIS
LIN {X 101.057,Y 53.813,Z 68.000,A 180.000,B 0.000,C 180.000} C_DIS
LIN {X 101.187,Y 53.638,Z 68.000,A 180.000,B 0.000,C 180.000} C_DIS
LIN {X 101.190,Y 53.634,Z 68.000,A 180.000,B 0.000,C 180.000} C_DIS
LIN {X 101.309,Y 53.455,Z 68.000,A 180.000,B 0.000,C 180.000} C_DIS
LIN {X 101.428,Y 53.277,Z 68.000,A 180.000,B 0.000,C 180.000} C_DIS
LIN {X 101.545,Y 53.098,Z 68.000,A 180.000,B 0.000,C 180.000} C_DIS
LIN {X 101.545,Y 53.098,Z 68.000,A 180.000,B 0.000,C 180.000} C_DIS
LIN {X 101.649,Y 52.919,Z 68.000,A 180.000,B 0.000,C 180.000} C_DIS
LIN {X 101.752,Y 52.740,Z 68.000,A 180.000,B 0.000,C 180.000} C_DIS
LIN {X 101.855,Y 52.562,Z 68.000,A 180.000,B 0.000,C 180.000} C_DIS
LIN {X 101.902,Y 52.473,Z 68.000,A 180.000,B 0.000,C 180.000} C_DIS
LIN {X 101.947,Y 52.383,Z 68.000,A 180.000,B 0.000,C 180.000} C_DIS
LIN {X 102.124,Y 52.025,Z 68.000,A 180.000,B 0.000,C 180.000} C_DIS
LIN {X 102.207,Y 51.847,Z 68.000,A 180.000,B 0.000,C 180.000} C_DIS
LIN {X 102.357,Y 51.489,Z 68.000,A 180.000,B 0.000,C 180.000} C_DIS
LIN {X 102.431,Y 51.310,Z 68.000,A 180.000,B 0.000,C 180.000} C_DIS
LIN {X 102.438,Y 51.291,Z 68.000,A 180.000,B 0.000,C 180.000} C_DIS
LIN {X 102.495,Y 51.131,Z 68.000,A 180.000,B 0.000,C 180.000} C_DIS
LIN {X 102.619,Y 50.774,Z 68.000,A 180.000,B 0.000,C 180.000} C_DIS
LIN {X 102.676,Y 50.595,Z 68.000,A 180.000,B 0.000,C 180.000} C_DIS
LIN {X 102.796,Y 50.163,Z 68.000,A 180.000,B 0.000,C 180.000} C_DIS
LIN {X 102.824,Y 50.059,Z 68.000,A 180.000,B 0.000,C 180.000} C_DIS
LIN {X 102.865,Y 49.880,Z 68.000,A 180.000,B 0.000,C 180.000} C_DIS
LIN {X 102.940,Y 49.523,Z 68.000,A 180.000,B 0.000,C 180.000} C_DIS
LIN {X 102.975,Y 49.350,Z 68.000,A 180.000,B 0.000,C 180.000} C_DIS
LIN {X 102.976,Y 49.344,Z 68.000,A 180.000,B 0.000,C 180.000} C_DIS
LIN {X 103.002,Y 49.165,Z 68.000,A 180.000,B 0.000,C 180.000} C_DIS
LIN {X 103.055,Y 48.807,Z 68.000,A 180.000,B 0.000,C 180.000} C_DIS
LIN {X 103.076,Y 48.629,Z 68.000,A 180.000,B 0.000,C 180.000} C_DIS
LIN {X 103.105,Y 48.271,Z 68.000,A 180.000,B 0.000,C 180.000} C_DIS
LIN {X 103.120,Y 48.092,Z 68.000,A 180.000,B 0.000,C 180.000} C_DIS
LIN {X 103.127,Y 47.914,Z 68.000,A 180.000,B 0.000,C 180.000} C_DIS
LIN {X 103.134,Y 47.556,Z 68.000,A 180.000,B 0.000,C 180.000} C_DIS
LIN {X 103.136,Y 47.377,Z 68.000,A 180.000,B 0.000,C 180.000} C_DIS
LIN {X 103.130,Y 47.198,Z 68.000,A 180.000,B 0.000,C 180.000} C_DIS
LIN {X 103.114,Y 46.841,Z 68.000,A 180.000,B 0.000,C 180.000} C_DIS
LIN {X 103.103,Y 46.662,Z 68.000,A 180.000,B 0.000,C 180.000} C_DIS
LIN {X 103.085,Y 46.483,Z 68.000,A 180.000,B 0.000,C 180.000} C_DIS
LIN {X 103.047,Y 46.126,Z 68.000,A 180.000,B 0.000,C 180.000} C_DIS
LIN {X 103.021,Y 45.947,Z 68.000,A 180.000,B 0.000,C 180.000} C_DIS
LIN {X 102.961,Y 45.590,Z 68.000,A 180.000,B 0.000,C 180.000} C_DIS
LIN {X 102.930,Y 45.411,Z 68.000,A 180.000,B 0.000,C 180.000} C_DIS
LIN {X 102.890,Y 45.232,Z 68.000,A 180.000,B 0.000,C 180.000} C_DIS
LIN {X 102.796,Y 44.834,Z 68.000,A 180.000,B 0.000,C 180.000} C_DIS
LIN {X 102.760,Y 44.696,Z 68.000,A 180.000,B 0.000,C 180.000} C_DIS
LIN {X 102.706,Y 44.517,Z 68.000,A 180.000,B 0.000,C 180.000} C_DIS
LIN {X 102.617,Y 44.222,Z 68.000,A 180.000,B 0.000,C 180.000} C_DIS
LIN {X 102.598,Y 44.159,Z 68.000,A 180.000,B 0.000,C 180.000} C_DIS
LIN {X 102.536,Y 43.981,Z 68.000,A 180.000,B 0.000,C 180.000} C_DIS
LIN {X 102.402,Y 43.623,Z 68.000,A 180.000,B 0.000,C 180.000} C_DIS
LIN {X 102.333,Y 43.444,Z 68.000,A 180.000,B 0.000,C 180.000} C_DIS
LIN {X 102.260,Y 43.278,Z 68.000,A 180.000,B 0.000,C 180.000} C_DIS
LIN {X 102.174,Y 43.087,Z 68.000,A 180.000,B 0.000,C 180.000} C_DIS
LIN {X 102.094,Y 42.908,Z 68.000,A 180.000,B 0.000,C 180.000} C_DIS
LIN {X 102.081,Y 42.879,Z 68.000,A 180.000,B 0.000,C 180.000} C_DIS
LIN {X 102.004,Y 42.729,Z 68.000,A 180.000,B 0.000,C 180.000} C_DIS
LIN {X 101.817,Y 42.372,Z 68.000,A 180.000,B 0.000,C 180.000} C_DIS
LIN {X 101.723,Y 42.203,Z 68.000,A 180.000,B 0.000,C 180.000} C_DIS
LIN {X 101.500,Y 41.835,Z 68.000,A 180.000,B 0.000,C 180.000} C_DIS
LIN {X 101.388,Y 41.657,Z 68.000,A 180.000,B 0.000,C 180.000} C_DIS
LIN {X 101.366,Y 41.625,Z 68.000,A 180.000,B 0.000,C 180.000} C_DIS
LIN {X 101.139,Y 41.299,Z 68.000,A 180.000,B 0.000,C 180.000} C_DIS
LIN {X 101.011,Y 41.120,Z 68.000,A 180.000,B 0.000,C 180.000} C_DIS
LIN {X 101.008,Y 41.117,Z 68.000,A 180.000,B 0.000,C 180.000} C_DIS
LIN {X 100.870,Y 40.942,Z 68.000,A 180.000,B 0.000,C 180.000} C_DIS
LIN {X 100.728,Y 40.763,Z 68.000,A 180.000,B 0.000,C 180.000} C_DIS
LIN {X 100.651,Y 40.666,Z 68.000,A 180.000,B 0.000,C 180.000} C_DIS
LIN {X 100.581,Y 40.584,Z 68.000,A 180.000,B 0.000,C 180.000} C_DIS
LIN {X 100.472,Y 40.463,Z 68.000,A 180.000,B 0.000,C 180.000} C_DIS
LIN {X 100.259,Y 40.226,Z 68.000,A 180.000,B 0.000,C 180.000} C_DIS
LIN {X 100.114,Y 40.074,Z 68.000,A 180.000,B 0.000,C 180.000} C_DIS
LIN {X 99.757,Y 39.725,Z 68.000,A 180.000,B 0.000,C 180.000} C_DIS
LIN {X 99.721,Y 39.690,Z 68.000,A 180.000,B 0.000,C 180.000} C_DIS
LIN {X 99.578,Y 39.563,Z 68.000,A 180.000,B 0.000,C 180.000} C_DIS
LIN {X 99.310,Y 39.333,Z 68.000,A 180.000,B 0.000,C 180.000} C_DIS
LIN {X 99.221,Y 39.256,Z 68.000,A 180.000,B 0.000,C 180.000} C_DIS
LIN {X 99.091,Y 39.154,Z 68.000,A 180.000,B 0.000,C 180.000} C_DIS
LIN {X 98.855,Y 38.975,Z 68.000,A 180.000,B 0.000,C 180.000} C_DIS
LIN {X 98.684,Y 38.846,Z 68.000,A 180.000,B 0.000,C 180.000} C_DIS
LIN {X 98.614,Y 38.796,Z 68.000,A 180.000,B 0.000,C 180.000} C_DIS
LIN {X 98.505,Y 38.724,Z 68.000,A 180.000,B 0.000,C 180.000} C_DIS
LIN {X 98.327,Y 38.606,Z 68.000,A 180.000,B 0.000,C 180.000} C_DIS
LIN {X 98.148,Y 38.487,Z 68.000,A 180.000,B 0.000,C 180.000} C_DIS
LIN {X 98.071,Y 38.439,Z 68.000,A 180.000,B 0.000,C 180.000} C_DIS
LIN {X 97.969,Y 38.380,Z 68.000,A 180.000,B 0.000,C 180.000} C_DIS
LIN {X 97.612,Y 38.174,Z 68.000,A 180.000,B 0.000,C 180.000} C_DIS
LIN {X 97.440,Y 38.081,Z 68.000,A 180.000,B 0.000,C 180.000} C_DIS
LIN {X 97.075,Y 37.900,Z 68.000,A 180.000,B 0.000,C 180.000} C_DIS
LIN {X 96.897,Y 37.814,Z 68.000,A 180.000,B 0.000,C 180.000} C_DIS
LIN {X 96.718,Y 37.739,Z 68.000,A 180.000,B 0.000,C 180.000} C_DIS
LIN {X 96.539,Y 37.664,Z 68.000,A 180.000,B 0.000,C 180.000} C_DIS
LIN {X 96.360,Y 37.589,Z 68.000,A 180.000,B 0.000,C 180.000} C_DIS
LIN {X 96.245,Y 37.545,Z 68.000,A 180.000,B 0.000,C 180.000} C_DIS
LIN {X 96.181,Y 37.523,Z 68.000,A 180.000,B 0.000,C 180.000} C_DIS
LIN {X 95.824,Y 37.399,Z 68.000,A 180.000,B 0.000,C 180.000} C_DIS
LIN {X 95.731,Y 37.366,Z 68.000,A 180.000,B 0.000,C 180.000} C_DIS
LIN {X 95.645,Y 37.339,Z 68.000,A 180.000,B 0.000,C 180.000} C_DIS
LIN {X 95.466,Y 37.289,Z 68.000,A 180.000,B 0.000,C 180.000} C_DIS
LIN {X 95.103,Y 37.187,Z 68.000,A 180.000,B 0.000,C 180.000} C_DIS
LIN {X 94.930,Y 37.146,Z 68.000,A 180.000,B 0.000,C 180.000} C_DIS
LIN {X 94.573,Y 37.070,Z 68.000,A 180.000,B 0.000,C 180.000} C_DIS
LIN {X 94.394,Y 37.033,Z 68.000,A 180.000,B 0.000,C 180.000} C_DIS
LIN {X 94.240,Y 37.009,Z 68.000,A 180.000,B 0.000,C 180.000} C_DIS
LIN {X 93.857,Y 36.952,Z 68.000,A 180.000,B 0.000,C 180.000} C_DIS
LIN {X 93.679,Y 36.929,Z 68.000,A 180.000,B 0.000,C 180.000} C_DIS
LIN {X 93.500,Y 36.914,Z 68.000,A 180.000,B 0.000,C 180.000} C_DIS
LIN {X 93.142,Y 36.884,Z 68.000,A 180.000,B 0.000,C 180.000} C_DIS
LIN {X 92.964,Y 36.874,Z 68.000,A 180.000,B 0.000,C 180.000} C_DIS
LIN {X 92.606,Y 36.867,Z 68.000,A 180.000,B 0.000,C 180.000} C_DIS
LIN {X 92.427,Y 36.864,Z 68.000,A 180.000,B 0.000,C 180.000} C_DIS
LIN {X 92.249,Y 36.868,Z 68.000,A 180.000,B 0.000,C 180.000} C_DIS
LIN {X 91.891,Y 36.883,Z 68.000,A 180.000,B 0.000,C 180.000} C_DIS
LIN {X 91.712,Y 36.892,Z 68.000,A 180.000,B 0.000,C 180.000} C_DIS
LIN {X 91.623,Y 36.901,Z 68.000,A 180.000,B 0.000,C 180.000} C_DIS
LIN {X 91.543,Y 36.909,Z 68.000,A 180.000,B 0.000,C 180.000} C_DIS
LIN {X 91.541,Y 36.909,Z 68.000,A 180.000,B 0.000,C 180.000} C_DIS
LIN {X 91.537,Y 36.902,Z 68.000,A 180.000,B 0.000,C 180.000} C_DIS
LIN {X 91.533,Y 36.894,Z 68.000,A 180.000,B 0.000,C 180.000} C_DIS
LIN {X 91.500,Y 36.830,Z 68.000,A 180.000,B 0.000,C 180.000} C_DIS
LIN {X 91.392,Y 36.651,Z 68.000,A 180.000,B 0.000,C 180.000} C_DIS
LIN {X 91.355,Y 36.595,Z 68.000,A 180.000,B 0.000,C 180.000} C_DIS
LIN {X 91.263,Y 36.472,Z 68.000,A 180.000,B 0.000,C 180.000} C_DIS
LIN {X 91.176,Y 36.368,Z 68.000,A 180.000,B 0.000,C 180.000} C_DIS
LIN {X 91.107,Y 36.294,Z 68.000,A 180.000,B 0.000,C 180.000} C_DIS
LIN {X 90.997,Y 36.186,Z 68.000,A 180.000,B 0.000,C 180.000} C_DIS
LIN {X 90.917,Y 36.115,Z 68.000,A 180.000,B 0.000,C 180.000} C_DIS
LIN {X 90.818,Y 36.036,Z 68.000,A 180.000,B 0.000,C 180.000} C_DIS
LIN {X 90.677,Y 35.936,Z 68.000,A 180.000,B 0.000,C 180.000} C_DIS
LIN {X 90.640,Y 35.912,Z 68.000,A 180.000,B 0.000,C 180.000} C_DIS
LIN {X 90.461,Y 35.809,Z 68.000,A 180.000,B 0.000,C 180.000} C_DIS
LIN {X 90.356,Y 35.757,Z 68.000,A 180.000,B 0.000,C 180.000} C_DIS
LIN {X 90.282,Y 35.724,Z 68.000,A 180.000,B 0.000,C 180.000} C_DIS
LIN {X 90.103,Y 35.656,Z 68.000,A 180.000,B 0.000,C 180.000} C_DIS
LIN {X 89.925,Y 35.603,Z 68.000,A 180.000,B 0.000,C 180.000} C_DIS
LIN {X 89.819,Y 35.578,Z 68.000,A 180.000,B 0.000,C 180.000} C_DIS
LIN {X 89.746,Y 35.564,Z 68.000,A 180.000,B 0.000,C 180.000} C_DIS
LIN {X 89.567,Y 35.539,Z 68.000,A 180.000,B 0.000,C 180.000} C_DIS
LIN {X 89.388,Y 35.526,Z 68.000,A 180.000,B 0.000,C 180.000} C_DIS
LIN {X 89.209,Y 35.526,Z 68.000,A 180.000,B 0.000,C 180.000} C_DIS
LIN {X 89.031,Y 35.540,Z 68.000,A 180.000,B 0.000,C 180.000} C_DIS
LIN {X 88.852,Y 35.566,Z 68.000,A 180.000,B 0.000,C 180.000} C_DIS
LIN {X 88.788,Y 35.578,Z 68.000,A 180.000,B 0.000,C 180.000} C_DIS
LIN {X 88.673,Y 35.605,Z 68.000,A 180.000,B 0.000,C 180.000} C_DIS
LIN {X 88.494,Y 35.659,Z 68.000,A 180.000,B 0.000,C 180.000} C_DIS
LIN {X 45.590,Y 50.133,Z 68.000,A 180.000,B 0.000,C 180.000} C_DIS
LIN {X 45.411,Y 50.194,Z 68.000,A 180.000,B 0.000,C 180.000} C_DIS
LIN {X 45.296,Y 50.238,Z 68.000,A 180.000,B 0.000,C 180.000} C_DIS
LIN {X 45.232,Y 50.265,Z 68.000,A 180.000,B 0.000,C 180.000} C_DIS
LIN {X 45.053,Y 50.353,Z 68.000,A 180.000,B 0.000,C 180.000} C_DIS
LIN {X 44.944,Y 50.416,Z 68.000,A 180.000,B 0.000,C 180.000} C_DIS
LIN {X 44.874,Y 50.461,Z 68.000,A 180.000,B 0.000,C 180.000} C_DIS
LIN {X 44.785,Y 50.522,Z 68.000,A 180.000,B 0.000,C 180.000} C_DIS
LIN {X 44.696,Y 50.590,Z 68.000,A 180.000,B 0.000,C 180.000} C_DIS
LIN {X 44.689,Y 50.595,Z 68.000,A 180.000,B 0.000,C 180.000} C_DIS
LIN {X 44.603,Y 50.667,Z 68.000,A 180.000,B 0.000,C 180.000} C_DIS
LIN {X 44.517,Y 50.746,Z 68.000,A 180.000,B 0.000,C 180.000} C_DIS
LIN {X 44.488,Y 50.774,Z 68.000,A 180.000,B 0.000,C 180.000} C_DIS
LIN {X 44.410,Y 50.855,Z 68.000,A 180.000,B 0.000,C 180.000} C_DIS
LIN {X 44.338,Y 50.936,Z 68.000,A 180.000,B 0.000,C 180.000} C_DIS
LIN {X 44.325,Y 50.953,Z 68.000,A 180.000,B 0.000,C 180.000} C_DIS
LIN {X 44.254,Y 51.042,Z 68.000,A 180.000,B 0.000,C 180.000} C_DIS
LIN {X 44.189,Y 51.131,Z 68.000,A 180.000,B 0.000,C 180.000} C_DIS
LIN {X 44.159,Y 51.176,Z 68.000,A 180.000,B 0.000,C 180.000} C_DIS
LIN {X 44.077,Y 51.310,Z 68.000,A 180.000,B 0.000,C 180.000} C_DIS
LIN {X 43.984,Y 51.489,Z 68.000,A 180.000,B 0.000,C 180.000} C_DIS
LIN {X 43.981,Y 51.497,Z 68.000,A 180.000,B 0.000,C 180.000} C_DIS
LIN {X 43.909,Y 51.668,Z 68.000,A 180.000,B 0.000,C 180.000} C_DIS
LIN {X 43.849,Y 51.847,Z 68.000,A 180.000,B 0.000,C 180.000} C_DIS
LIN {X 43.804,Y 52.025,Z 68.000,A 180.000,B 0.000,C 180.000} C_DIS
LIN {X 43.802,Y 52.035,Z 68.000,A 180.000,B 0.000,C 180.000} C_DIS
LIN {X 43.772,Y 52.204,Z 68.000,A 180.000,B 0.000,C 180.000} C_DIS
LIN {X 43.754,Y 52.383,Z 68.000,A 180.000,B 0.000,C 180.000} C_DIS
LIN {X 43.748,Y 52.562,Z 68.000,A 180.000,B 0.000,C 180.000} C_DIS
LIN {X 43.756,Y 52.740,Z 68.000,A 180.000,B 0.000,C 180.000} C_DIS
LIN {X 43.776,Y 52.919,Z 68.000,A 180.000,B 0.000,C 180.000} C_DIS
LIN {X 43.802,Y 53.064,Z 68.000,A 180.000,B 0.000,C 180.000} C_DIS
LIN {X 43.809,Y 53.098,Z 68.000,A 180.000,B 0.000,C 180.000} C_DIS
LIN {X 43.856,Y 53.277,Z 68.000,A 180.000,B 0.000,C 180.000} C_DIS
LIN {X 43.916,Y 53.455,Z 68.000,A 180.000,B 0.000,C 180.000} C_DIS
LIN {X 47.391,Y 63.759,Z 68.000,A 180.000,B 0.000,C 180.000} C_DIS
LIN {X 50.248,Y 72.226,Z 68.000,A 180.000,B 0.000,C 180.000} C_DIS
LIN {X 50.311,Y 72.405,Z 68.000,A 180.000,B 0.000,C 180.000} C_DIS
LIN {X 50.388,Y 72.584,Z 68.000,A 180.000,B 0.000,C 180.000} C_DIS
LIN {X 50.416,Y 72.640,Z 68.000,A 180.000,B 0.000,C 180.000} C_DIS
LIN {X 50.484,Y 72.763,Z 68.000,A 180.000,B 0.000,C 180.000} C_DIS
LIN {X 50.595,Y 72.936,Z 68.000,A 180.000,B 0.000,C 180.000} C_DIS
LIN {X 50.599,Y 72.941,Z 68.000,A 180.000,B 0.000,C 180.000} C_DIS
LIN {X 50.665,Y 73.031,Z 68.000,A 180.000,B 0.000,C 180.000} C_DIS
LIN {X 50.737,Y 73.120,Z 68.000,A 180.000,B 0.000,C 180.000} C_DIS
LIN {X 50.774,Y 73.162,Z 68.000,A 180.000,B 0.000,C 180.000} C_DIS
LIN {X 50.905,Y 73.299,Z 68.000,A 180.000,B 0.000,C 180.000} C_DIS
LIN {X 50.953,Y 73.343,Z 68.000,A 180.000,B 0.000,C 180.000} C_DIS
LIN {X 51.112,Y 73.478,Z 68.000,A 180.000,B 0.000,C 180.000} C_DIS
LIN {X 51.131,Y 73.493,Z 68.000,A 180.000,B 0.000,C 180.000} C_DIS
LIN {X 51.310,Y 73.616,Z 68.000,A 180.000,B 0.000,C 180.000} C_DIS
LIN {X 51.376,Y 73.656,Z 68.000,A 180.000,B 0.000,C 180.000} C_DIS
LIN {X 51.489,Y 73.719,Z 68.000,A 180.000,B 0.000,C 180.000} C_DIS
LIN {X 51.668,Y 73.803,Z 68.000,A 180.000,B 0.000,C 180.000} C_DIS
LIN {X 51.749,Y 73.835,Z 68.000,A 180.000,B 0.000,C 180.000} C_DIS
LIN {X 51.847,Y 73.870,Z 68.000,A 180.000,B 0.000,C 180.000} C_DIS
LIN {X 52.025,Y 73.923,Z 68.000,A 180.000,B 0.000,C 180.000} C_DIS
LIN {X 52.204,Y 73.961,Z 68.000,A 180.000,B 0.000,C 180.000} C_DIS
LIN {X 52.383,Y 73.987,Z 68.000,A 180.000,B 0.000,C 180.000} C_DIS
LIN {X 52.562,Y 73.999,Z 68.000,A 180.000,B 0.000,C 180.000} C_DIS
LIN {X 52.740,Y 73.998,Z 68.000,A 180.000,B 0.000,C 180.000} C_DIS
LIN {X 52.919,Y 73.985,Z 68.000,A 180.000,B 0.000,C 180.000} C_DIS
LIN {X 53.098,Y 73.958,Z 68.000,A 180.000,B 0.000,C 180.000} C_DIS
LIN {X 53.277,Y 73.918,Z 68.000,A 180.000,B 0.000,C 180.000} C_DIS
LIN {X 53.455,Y 73.864,Z 68.000,A 180.000,B 0.000,C 180.000} C_DIS
LIN {X 76.321,Y 66.150,Z 68.000,A 180.000,B 0.000,C 180.000} C_DIS
; Link Move Starts
LIN {X 76.620,Y 66.049,Z 68.000,A 180.000,B 0.000,C 180.000} C_DIS
LIN {X 76.918,Y 65.949,Z 67.999,A 180.000,B 0.000,C 180.000} C_DIS
LIN {X 77.217,Y 65.848,Z 67.998,A 180.000,B 0.000,C 180.000} C_DIS
LIN {X 77.515,Y 65.747,Z 67.996,A 180.000,B 0.000,C 180.000} C_DIS
LIN {X 77.814,Y 65.647,Z 67.994,A 180.000,B 0.000,C 180.000} C_DIS
LIN {X 78.112,Y 65.546,Z 67.991,A 180.000,B 0.000,C 180.000} C_DIS
LIN {X 78.411,Y 65.445,Z 67.988,A 180.000,B 0.000,C 180.000} C_DIS
LIN {X 78.709,Y 65.344,Z 67.985,A 180.000,B 0.000,C 180.000} C_DIS
LIN {X 79.008,Y 65.244,Z 67.981,A 180.000,B 0.000,C 180.000} C_DIS
LIN {X 79.306,Y 65.143,Z 67.977,A 180.000,B 0.000,C 180.000} C_DIS
LIN {X 79.604,Y 65.042,Z 67.972,A 180.000,B 0.000,C 180.000} C_DIS
LIN {X 79.754,Y 64.992,Z 67.969,A 180.000,B 0.000,C 180.000} C_DIS
LIN {X 79.903,Y 64.942,Z 67.967,A 180.000,B 0.000,C 180.000} C_DIS
LIN {X 80.052,Y 64.891,Z 67.964,A 180.000,B 0.000,C 180.000} C_DIS
LIN {X 80.201,Y 64.841,Z 67.961,A 180.000,B 0.000,C 180.000} C_DIS
LIN {X 80.351,Y 64.791,Z 67.959,A 180.000,B 0.000,C 180.000} C_DIS
LIN {X 80.500,Y 64.740,Z 67.956,A 180.000,B 0.000,C 180.000} C_DIS
LIN {X 80.649,Y 64.690,Z 67.952,A 180.000,B 0.000,C 180.000} C_DIS
LIN {X 80.798,Y 64.640,Z 67.949,A 180.000,B 0.000,C 180.000} C_DIS
LIN {X 80.948,Y 64.589,Z 67.946,A 180.000,B 0.000,C 180.000} C_DIS
LIN {X 81.097,Y 64.539,Z 67.943,A 180.000,B 0.000,C 180.000} C_DIS
LIN {X 81.246,Y 64.489,Z 67.939,A 180.000,B 0.000,C 180.000} C_DIS
LIN {X 81.395,Y 64.438,Z 67.936,A 180.000,B 0.000,C 180.000} C_DIS
LIN {X 81.545,Y 64.388,Z 67.932,A 180.000,B 0.000,C 180.000} C_DIS
LIN {X 81.694,Y 64.338,Z 67.928,A 180.000,B 0.000,C 180.000} C_DIS
LIN {X 81.843,Y 64.287,Z 67.925,A 180.000,B 0.000,C 180.000} C_DIS
LIN {X 81.992,Y 64.237,Z 67.921,A 180.000,B 0.000,C 180.000} C_DIS
LIN {X 82.141,Y 64.187,Z 67.917,A 180.000,B 0.000,C 180.000} C_DIS
LIN {X 82.291,Y 64.136,Z 67.913,A 180.000,B 0.000,C 180.000} C_DIS
LIN {X 82.440,Y 64.086,Z 67.909,A 180.000,B 0.000,C 180.000} C_DIS
LIN {X 82.589,Y 64.036,Z 67.905,A 180.000,B 0.000,C 180.000} C_DIS
LIN {X 82.738,Y 63.985,Z 67.900,A 180.000,B 0.000,C 180.000} C_DIS
LIN {X 82.888,Y 63.935,Z 67.896,A 180.000,B 0.000,C 180.000} C_DIS
LIN {X 83.037,Y 63.884,Z 67.892,A 180.000,B 0.000,C 180.000} C_DIS
LIN {X 83.186,Y 63.834,Z 67.887,A 180.000,B 0.000,C 180.000} C_DIS
LIN {X 83.335,Y 63.784,Z 67.883,A 180.000,B 0.000,C 180.000} C_DIS
LIN {X 83.485,Y 63.733,Z 67.878,A 180.000,B 0.000,C 180.000} C_DIS
LIN {X 83.634,Y 63.683,Z 67.873,A 180.000,B 0.000,C 180.000} C_DIS
LIN {X 83.783,Y 63.633,Z 67.869,A 180.000,B 0.000,C 180.000} C_DIS
LIN {X 83.932,Y 63.582,Z 67.864,A 180.000,B 0.000,C 180.000} C_DIS
LIN {X 84.082,Y 63.532,Z 67.859,A 180.000,B 0.000,C 180.000} C_DIS
LIN {X 84.231,Y 63.482,Z 67.854,A 180.000,B 0.000,C 180.000} C_DIS
LIN {X 84.305,Y 63.457,Z 67.851,A 180.000,B 0.000,C 180.000} C_DIS
LIN {X 84.380,Y 63.431,Z 67.849,A 180.000,B 0.000,C 180.000} C_DIS
LIN {X 84.455,Y 63.406,Z 67.846,A 180.000,B 0.000,C 180.000} C_DIS
LIN {X 84.529,Y 63.381,Z 67.844,A 180.000,B 0.000,C 180.000} C_DIS
LIN {X 84.604,Y 63.356,Z 67.841,A 180.000,B 0.000,C 180.000} C_DIS
LIN {X 84.679,Y 63.331,Z 67.839,A 180.000,B 0.000,C 180.000} C_DIS
LIN {X 84.753,Y 63.306,Z 67.836,A 180.000,B 0.000,C 180.000} C_DIS
LIN {X 84.902,Y 63.255,Z 67.831,A 180.000,B 0.000,C 180.000} C_DIS
LIN {X 85.052,Y 63.205,Z 67.825,A 180.000,B 0.000,C 180.000} C_DIS
LIN {X 85.201,Y 63.154,Z 67.820,A 180.000,B 0.000,C 180.000} C_DIS
LIN {X 85.350,Y 63.104,Z 67.815,A 180.000,B 0.000,C 180.000} C_DIS
LIN {X 85.499,Y 63.054,Z 67.809,A 180.000,B 0.000,C 180.000} C_DIS
LIN {X 85.574,Y 63.029,Z 67.807,A 180.000,B 0.000,C 180.000} C_DIS
LIN {X 85.723,Y 62.978,Z 67.801,A 180.000,B 0.000,C 180.000} C_DIS
LIN {X 85.947,Y 62.903,Z 67.793,A 180.000,B 0.000,C 180.000} C_DIS
LIN {X 86.096,Y 62.852,Z 67.787,A 180.000,B 0.000,C 180.000} C_DIS
LIN {X 86.171,Y 62.827,Z 67.785,A 180.000,B 0.000,C 180.000} C_DIS
LIN {X 86.320,Y 62.777,Z 67.779,A 180.000,B 0.000,C 180.000} C_DIS
LIN {X 86.544,Y 62.701,Z 67.771,A 180.000,B 0.000,C 180.000} C_DIS
LIN {X 86.693,Y 62.651,Z 67.765,A 180.000,B 0.000,C 180.000} C_DIS
LIN {X 86.768,Y 62.626,Z 67.763,A 180.000,B 0.000,C 180.000} C_DIS
LIN {X 86.917,Y 62.576,Z 67.757,A 180.000,B 0.000,C 180.000} C_DIS
LIN {X 87.141,Y 62.500,Z 67.749,A 180.000,B 0.000,C 180.000} C_DIS
LIN {X 87.290,Y 62.450,Z 67.743,A 180.000,B 0.000,C 180.000} C_DIS
LIN {X 87.365,Y 62.424,Z 67.741,A 180.000,B 0.000,C 180.000} C_DIS
LIN {X 87.514,Y 62.374,Z 67.735,A 180.000,B 0.000,C 180.000} C_DIS
LIN {X 87.738,Y 62.299,Z 67.727,A 180.000,B 0.000,C 180.000} C_DIS
LIN {X 87.887,Y 62.248,Z 67.721,A 180.000,B 0.000,C 180.000} C_DIS
LIN {X 87.962,Y 62.223,Z 67.719,A 180.000,B 0.000,C 180.000} C_DIS
LIN {X 88.111,Y 62.173,Z 67.713,A 180.000,B 0.000,C 180.000} C_DIS
LIN {X 88.559,Y 62.022,Z 67.697,A 180.000,B 0.000,C 180.000} C_DIS
LIN {X 88.708,Y 61.971,Z 67.691,A 180.000,B 0.000,C 180.000} C_DIS
LIN {X 89.156,Y 61.820,Z 67.675,A 180.000,B 0.000,C 180.000} C_DIS
LIN {X 89.305,Y 61.770,Z 67.669,A 180.000,B 0.000,C 180.000} C_DIS
LIN {X 89.827,Y 61.594,Z 67.650,A 180.000,B 0.000,C 180.000} C_DIS
LIN {X 90.275,Y 61.443,Z 67.633,A 180.000,B 0.000,C 180.000} C_DIS
LIN {X 90.424,Y 61.392,Z 67.628,A 180.000,B 0.000,C 180.000} C_DIS
LIN {X 90.872,Y 61.241,Z 67.611,A 180.000,B 0.000,C 180.000} C_DIS
LIN {X 91.021,Y 61.191,Z 67.606,A 180.000,B 0.000,C 180.000} C_DIS
LIN {X 91.693,Y 60.964,Z 67.581,A 180.000,B 0.000,C 180.000} C_DIS
LIN {X 92.737,Y 60.612,Z 67.543,A 180.000,B 0.000,C 180.000} C_DIS
LIN {X 93.483,Y 60.360,Z 67.515,A 180.000,B 0.000,C 180.000} C_DIS
LIN {X 96.468,Y 59.353,Z 67.405,A 180.000,B 0.000,C 180.000} C_DIS
LIN {X 96.543,Y 59.328,Z 67.402,A 180.000,B 0.000,C 180.000} C_DIS
LIN {X 96.616,Y 59.300,Z 67.400,A 180.000,B 0.000,C 180.000} C_DIS
LIN {X 96.689,Y 59.270,Z 67.397,A 180.000,B 0.000,C 180.000} C_DIS
LIN {X 96.761,Y 59.237,Z 67.394,A 180.000,B 0.000,C 180.000} C_DIS
LIN {X 96.832,Y 59.203,Z 67.391,A 180.000,B 0.000,C 180.000} C_DIS
LIN {X 96.901,Y 59.166,Z 67.389,A 180.000,B 0.000,C 180.000} C_DIS
LIN {X 96.970,Y 59.127,Z 67.386,A 180.000,B 0.000,C 180.000} C_DIS
LIN {X 97.037,Y 59.086,Z 67.383,A 180.000,B 0.000,C 180.000} C_DIS
LIN {X 97.103,Y 59.042,Z 67.380,A 180.000,B 0.000,C 180.000} C_DIS
LIN {X 97.167,Y 58.997,Z 67.378,A 180.000,B 0.000,C 180.000} C_DIS
LIN {X 97.230,Y 58.950,Z 67.375,A 180.000,B 0.000,C 180.000} C_DIS
LIN {X 97.291,Y 58.901,Z 67.372,A 180.000,B 0.000,C 180.000} C_DIS
LIN {X 97.351,Y 58.849,Z 67.369,A 180.000,B 0.000,C 180.000} C_DIS
LIN {X 97.409,Y 58.796,Z 67.367,A 180.000,B 0.000,C 180.000} C_DIS
LIN {X 97.466,Y 58.741,Z 67.364,A 180.000,B 0.000,C 180.000} C_DIS
LIN {X 97.521,Y 58.685,Z 67.361,A 180.000,B 0.000,C 180.000} C_DIS
LIN {X 97.574,Y 58.627,Z 67.358,A 180.000,B 0.000,C 180.000} C_DIS
LIN {X 97.625,Y 58.567,Z 67.356,A 180.000,B 0.000,C 180.000} C_DIS
LIN {X 97.674,Y 58.505,Z 67.353,A 180.000,B 0.000,C 180.000} C_DIS
LIN {X 97.721,Y 58.442,Z 67.350,A 180.000,B 0.000,C 180.000} C_DIS
LIN {X 97.766,Y 58.377,Z 67.347,A 180.000,B 0.000,C 180.000} C_DIS
LIN {X 97.809,Y 58.312,Z 67.345,A 180.000,B 0.000,C 180.000} C_DIS
LIN {X 97.850,Y 58.244,Z 67.342,A 180.000,B 0.000,C 180.000} C_DIS
LIN {X 97.889,Y 58.176,Z 67.339,A 180.000,B 0.000,C 180.000} C_DIS
LIN {X 97.926,Y 58.106,Z 67.336,A 180.000,B 0.000,C 180.000} C_DIS
LIN {X 97.961,Y 58.035,Z 67.334,A 180.000,B 0.000,C 180.000} C_DIS
LIN {X 97.993,Y 57.964,Z 67.331,A 180.000,B 0.000,C 180.000} C_DIS
LIN {X 98.023,Y 57.891,Z 67.328,A 180.000,B 0.000,C 180.000} C_DIS
LIN {X 98.051,Y 57.817,Z 67.325,A 180.000,B 0.000,C 180.000} C_DIS
LIN {X 98.076,Y 57.742,Z 67.323,A 180.000,B 0.000,C 180.000} C_DIS
LIN {X 98.099,Y 57.667,Z 67.320,A 180.000,B 0.000,C 180.000} C_DIS
LIN {X 98.119,Y 57.591,Z 67.317,A 180.000,B 0.000,C 180.000} C_DIS
LIN {X 98.138,Y 57.514,Z 67.314,A 180.000,B 0.000,C 180.000} C_DIS
LIN {X 98.153,Y 57.437,Z 67.312,A 180.000,B 0.000,C 180.000} C_DIS
LIN {X 98.170,Y 57.341,Z 67.308,A 180.000,B 0.000,C 180.000} C_DIS
LIN {X 98.182,Y 57.245,Z 67.305,A 180.000,B 0.000,C 180.000} C_DIS
LIN {X 98.187,Y 57.191,Z 67.303,A 180.000,B 0.000,C 180.000} C_DIS
LIN {X 98.189,Y 57.164,Z 67.303,A 180.000,B 0.000,C 180.000} C_DIS
LIN {X 98.190,Y 57.150,Z 67.302,A 180.000,B 0.000,C 180.000} C_DIS
LIN {X 98.191,Y 57.146,Z 67.302,A 180.000,B 0.000,C 180.000} C_DIS
LIN {X 98.192,Y 57.143,Z 67.302,A 180.000,B 0.000,C 180.000} C_DIS
LIN {X 98.199,Y 57.139,Z 67.302,A 180.000,B 0.000,C 180.000} C_DIS
LIN {X 98.292,Y 57.085,Z 67.298,A 180.000,B 0.000,C 180.000} C_DIS
LIN {X 98.429,Y 57.007,Z 67.293,A 180.000,B 0.000,C 180.000} C_DIS
LIN {X 98.497,Y 56.968,Z 67.290,A 180.000,B 0.000,C 180.000} C_DIS
LIN {X 98.566,Y 56.929,Z 67.287,A 180.000,B 0.000,C 180.000} C_DIS
LIN {X 98.631,Y 56.889,Z 67.285,A 180.000,B 0.000,C 180.000} C_DIS
LIN {X 98.694,Y 56.848,Z 67.282,A 180.000,B 0.000,C 180.000} C_DIS
LIN {X 98.887,Y 56.721,Z 67.274,A 180.000,B 0.000,C 180.000} C_DIS
LIN {X 99.018,Y 56.635,Z 67.269,A 180.000,B 0.000,C 180.000} C_DIS
LIN {X 99.084,Y 56.591,Z 67.266,A 180.000,B 0.000,C 180.000} C_DIS
LIN {X 99.148,Y 56.550,Z 67.263,A 180.000,B 0.000,C 180.000} C_DIS
LIN {X 99.210,Y 56.507,Z 67.260,A 180.000,B 0.000,C 180.000} C_DIS
LIN {X 99.272,Y 56.462,Z 67.258,A 180.000,B 0.000,C 180.000} C_DIS
LIN {X 99.333,Y 56.416,Z 67.255,A 180.000,B 0.000,C 180.000} C_DIS
LIN {X 99.458,Y 56.321,Z 67.250,A 180.000,B 0.000,C 180.000} C_DIS
LIN {X 99.646,Y 56.180,Z 67.241,A 180.000,B 0.000,C 180.000} C_DIS
LIN {X 99.708,Y 56.133,Z 67.239,A 180.000,B 0.000,C 180.000} C_DIS
LIN {X 99.770,Y 56.085,Z 67.236,A 180.000,B 0.000,C 180.000} C_DIS
LIN {X 99.829,Y 56.035,Z 67.233,A 180.000,B 0.000,C 180.000} C_DIS
LIN {X 99.947,Y 55.935,Z 67.228,A 180.000,B 0.000,C 180.000} C_DIS
LIN {X 100.124,Y 55.783,Z 67.220,A 180.000,B 0.000,C 180.000} C_DIS
LIN {X 100.242,Y 55.683,Z 67.214,A 180.000,B 0.000,C 180.000} C_DIS
LIN {X 100.300,Y 55.631,Z 67.212,A 180.000,B 0.000,C 180.000} C_DIS
LIN {X 100.357,Y 55.578,Z 67.209,A 180.000,B 0.000,C 180.000} C_DIS
LIN {X 100.413,Y 55.524,Z 67.206,A 180.000,B 0.000,C 180.000} C_DIS
LIN {X 100.468,Y 55.470,Z 67.204,A 180.000,B 0.000,C 180.000} C_DIS
LIN {X 100.524,Y 55.415,Z 67.201,A 180.000,B 0.000,C 180.000} C_DIS
LIN {X 100.581,Y 55.361,Z 67.198,A 180.000,B 0.000,C 180.000} C_DIS
LIN {X 100.637,Y 55.306,Z 67.195,A 180.000,B 0.000,C 180.000} C_DIS
LIN {X 100.694,Y 55.251,Z 67.193,A 180.000,B 0.000,C 180.000} C_DIS
LIN {X 100.750,Y 55.196,Z 67.190,A 180.000,B 0.000,C 180.000} C_DIS
LIN {X 100.804,Y 55.142,Z 67.187,A 180.000,B 0.000,C 180.000} C_DIS
LIN {X 100.857,Y 55.085,Z 67.185,A 180.000,B 0.000,C 180.000} C_DIS
LIN {X 100.909,Y 55.028,Z 67.182,A 180.000,B 0.000,C 180.000} C_DIS
LIN {X 100.960,Y 54.971,Z 67.179,A 180.000,B 0.000,C 180.000} C_DIS
LIN {X 101.013,Y 54.912,Z 67.177,A 180.000,B 0.000,C 180.000} C_DIS
LIN {X 101.066,Y 54.854,Z 67.174,A 180.000,B 0.000,C 180.000} C_DIS
LIN {X 101.118,Y 54.795,Z 67.171,A 180.000,B 0.000,C 180.000} C_DIS
LIN {X 101.171,Y 54.737,Z 67.169,A 180.000,B 0.000,C 180.000} C_DIS
LIN {X 101.223,Y 54.679,Z 67.166,A 180.000,B 0.000,C 180.000} C_DIS
LIN {X 101.274,Y 54.621,Z 67.164,A 180.000,B 0.000,C 180.000} C_DIS
LIN {X 101.371,Y 54.501,Z 67.159,A 180.000,B 0.000,C 180.000} C_DIS
LIN {X 101.420,Y 54.439,Z 67.156,A 180.000,B 0.000,C 180.000} C_DIS
LIN {X 101.469,Y 54.378,Z 67.154,A 180.000,B 0.000,C 180.000} C_DIS
LIN {X 101.517,Y 54.316,Z 67.151,A 180.000,B 0.000,C 180.000} C_DIS
LIN {X 101.566,Y 54.254,Z 67.149,A 180.000,B 0.000,C 180.000} C_DIS
LIN {X 101.663,Y 54.132,Z 67.144,A 180.000,B 0.000,C 180.000} C_DIS
LIN {X 101.757,Y 54.008,Z 67.139,A 180.000,B 0.000,C 180.000} C_DIS
LIN {X 101.846,Y 53.879,Z 67.134,A 180.000,B 0.000,C 180.000} C_DIS
LIN {X 101.935,Y 53.750,Z 67.129,A 180.000,B 0.000,C 180.000} C_DIS
LIN {X 102.024,Y 53.621,Z 67.125,A 180.000,B 0.000,C 180.000} C_DIS
LIN {X 102.113,Y 53.492,Z 67.120,A 180.000,B 0.000,C 180.000} C_DIS
LIN {X 102.195,Y 53.360,Z 67.116,A 180.000,B 0.000,C 180.000} C_DIS
LIN {X 102.356,Y 53.091,Z 67.107,A 180.000,B 0.000,C 180.000} C_DIS
LIN {X 102.437,Y 52.956,Z 67.102,A 180.000,B 0.000,C 180.000} C_DIS
LIN {X 102.515,Y 52.821,Z 67.098,A 180.000,B 0.000,C 180.000} C_DIS
LIN {X 102.587,Y 52.683,Z 67.094,A 180.000,B 0.000,C 180.000} C_DIS
LIN {X 102.659,Y 52.543,Z 67.090,A 180.000,B 0.000,C 180.000} C_DIS
LIN {X 102.731,Y 52.403,Z 67.086,A 180.000,B 0.000,C 180.000} C_DIS
LIN {X 102.803,Y 52.265,Z 67.082,A 180.000,B 0.000,C 180.000} C_DIS
LIN {X 102.868,Y 52.123,Z 67.078,A 180.000,B 0.000,C 180.000} C_DIS
LIN {X 102.931,Y 51.979,Z 67.074,A 180.000,B 0.000,C 180.000} C_DIS
LIN {X 102.994,Y 51.835,Z 67.071,A 180.000,B 0.000,C 180.000} C_DIS
LIN {X 103.057,Y 51.691,Z 67.067,A 180.000,B 0.000,C 180.000} C_DIS
LIN {X 103.118,Y 51.547,Z 67.063,A 180.000,B 0.000,C 180.000} C_DIS
LIN {X 103.172,Y 51.399,Z 67.060,A 180.000,B 0.000,C 180.000} C_DIS
LIN {X 103.226,Y 51.251,Z 67.057,A 180.000,B 0.000,C 180.000} C_DIS
LIN {X 103.280,Y 51.103,Z 67.053,A 180.000,B 0.000,C 180.000} C_DIS
LIN {X 103.333,Y 50.955,Z 67.050,A 180.000,B 0.000,C 180.000} C_DIS
LIN {X 103.381,Y 50.806,Z 67.047,A 180.000,B 0.000,C 180.000} C_DIS
LIN {X 103.425,Y 50.656,Z 67.044,A 180.000,B 0.000,C 180.000} C_DIS
LIN {X 103.469,Y 50.505,Z 67.041,A 180.000,B 0.000,C 180.000} C_DIS
LIN {X 103.513,Y 50.354,Z 67.038,A 180.000,B 0.000,C 180.000} C_DIS
LIN {X 103.555,Y 50.203,Z 67.035,A 180.000,B 0.000,C 180.000} C_DIS
LIN {X 103.590,Y 50.050,Z 67.033,A 180.000,B 0.000,C 180.000} C_DIS
LIN {X 103.625,Y 49.896,Z 67.030,A 180.000,B 0.000,C 180.000} C_DIS
LIN {X 103.659,Y 49.742,Z 67.028,A 180.000,B 0.000,C 180.000} C_DIS
LIN {X 103.722,Y 49.434,Z 67.023,A 180.000,B 0.000,C 180.000} C_DIS
LIN {X 103.771,Y 49.123,Z 67.019,A 180.000,B 0.000,C 180.000} C_DIS
LIN {X 103.818,Y 48.812,Z 67.015,A 180.000,B 0.000,C 180.000} C_DIS
LIN {X 103.848,Y 48.499,Z 67.012,A 180.000,B 0.000,C 180.000} C_DIS
LIN {X 103.876,Y 48.185,Z 67.008,A 180.000,B 0.000,C 180.000} C_DIS
LIN {X 103.890,Y 47.871,Z 67.006,A 180.000,B 0.000,C 180.000} C_DIS
LIN {X 103.897,Y 47.556,Z 67.004,A 180.000,B 0.000,C 180.000} C_DIS
LIN {X 103.897,Y 47.241,Z 67.002,A 180.000,B 0.000,C 180.000} C_DIS
LIN {X 103.884,Y 46.926,Z 67.001,A 180.000,B 0.000,C 180.000} C_DIS
LIN {X 103.868,Y 46.612,Z 67.000,A 180.000,B 0.000,C 180.000} C_DIS
LIN {X 103.836,Y 46.305,Z 67.000,A 180.000,B 0.000,C 180.000} C_DIS
; Cutting Move Starts
LIN {X 103.817,Y 46.126,Z 67.000,A 180.000,B 0.000,C 180.000} C_DIS
LIN {X 103.797,Y 45.947,Z 67.000,A 180.000,B 0.000,C 180.000} C_DIS
LIN {X 103.768,Y 45.768,Z 67.000,A 180.000,B 0.000,C 180.000} C_DIS
LIN {X 103.690,Y 45.310,Z 67.000,A 180.000,B 0.000,C 180.000} C_DIS
LIN {X 103.675,Y 45.232,Z 67.000,A 180.000,B 0.000,C 180.000} C_DIS
LIN {X 103.634,Y 45.053,Z 67.000,A 180.000,B 0.000,C 180.000} C_DIS
LIN {X 103.550,Y 44.696,Z 67.000,A 180.000,B 0.000,C 180.000} C_DIS
LIN {X 103.511,Y 44.536,Z 67.000,A 180.000,B 0.000,C 180.000} C_DIS
LIN {X 103.506,Y 44.517,Z 67.000,A 180.000,B 0.000,C 180.000} C_DIS
LIN {X 103.452,Y 44.338,Z 67.000,A 180.000,B 0.000,C 180.000} C_DIS
LIN {X 103.332,Y 43.942,Z 67.000,A 180.000,B 0.000,C 180.000} C_DIS
LIN {X 103.286,Y 43.802,Z 67.000,A 180.000,B 0.000,C 180.000} C_DIS
LIN {X 103.220,Y 43.623,Z 67.000,A 180.000,B 0.000,C 180.000} C_DIS
LIN {X 103.086,Y 43.266,Z 67.000,A 180.000,B 0.000,C 180.000} C_DIS
LIN {X 103.013,Y 43.087,Z 67.000,A 180.000,B 0.000,C 180.000} C_DIS
LIN {X 102.796,Y 42.601,Z 67.000,A 180.000,B 0.000,C 180.000} C_DIS
LIN {X 102.773,Y 42.550,Z 67.000,A 180.000,B 0.000,C 180.000} C_DIS
LIN {X 102.681,Y 42.372,Z 67.000,A 180.000,B 0.000,C 180.000} C_DIS
LIN {X 102.494,Y 42.014,Z 67.000,A 180.000,B 0.000,C 180.000} C_DIS
LIN {X 102.438,Y 41.909,Z 67.000,A 180.000,B 0.000,C 180.000} C_DIS
LIN {X 102.396,Y 41.835,Z 67.000,A 180.000,B 0.000,C 180.000} C_DIS
LIN {X 102.260,Y 41.611,Z 67.000,A 180.000,B 0.000,C 180.000} C_DIS
LIN {X 102.179,Y 41.478,Z 67.000,A 180.000,B 0.000,C 180.000} C_DIS
LIN {X 102.081,Y 41.317,Z 67.000,A 180.000,B 0.000,C 180.000} C_DIS
LIN {X 102.069,Y 41.299,Z 67.000,A 180.000,B 0.000,C 180.000} C_DIS
LIN {X 101.947,Y 41.120,Z 67.000,A 180.000,B 0.000,C 180.000} C_DIS
LIN {X 101.699,Y 40.763,Z 67.000,A 180.000,B 0.000,C 180.000} C_DIS
LIN {X 101.563,Y 40.584,Z 67.000,A 180.000,B 0.000,C 180.000} C_DIS
LIN {X 101.280,Y 40.226,Z 67.000,A 180.000,B 0.000,C 180.000} C_DIS
LIN {X 101.187,Y 40.113,Z 67.000,A 180.000,B 0.000,C 180.000} C_DIS
LIN {X 101.128,Y 40.048,Z 67.000,A 180.000,B 0.000,C 180.000} C_DIS
LIN {X 100.806,Y 39.690,Z 67.000,A 180.000,B 0.000,C 180.000} C_DIS
LIN {X 100.651,Y 39.528,Z 67.000,A 180.000,B 0.000,C 180.000} C_DIS
LIN {X 100.268,Y 39.154,Z 67.000,A 180.000,B 0.000,C 180.000} C_DIS
LIN {X 100.114,Y 39.015,Z 67.000,A 180.000,B 0.000,C 180.000} C_DIS
LIN {X 99.757,Y 38.707,Z 67.000,A 180.000,B 0.000,C 180.000} C_DIS
LIN {X 99.650,Y 38.618,Z 67.000,A 180.000,B 0.000,C 180.000} C_DIS
LIN {X 99.578,Y 38.562,Z 67.000,A 180.000,B 0.000,C 180.000} C_DIS
LIN {X 99.180,Y 38.260,Z 67.000,A 180.000,B 0.000,C 180.000} C_DIS
LIN {X 99.042,Y 38.161,Z 67.000,A 180.000,B 0.000,C 180.000} C_DIS
LIN {X 98.921,Y 38.081,Z 67.000,A 180.000,B 0.000,C 180.000} C_DIS
LIN {X 98.652,Y 37.902,Z 67.000,A 180.000,B 0.000,C 180.000} C_DIS
LIN {X 98.505,Y 37.807,Z 67.000,A 180.000,B 0.000,C 180.000} C_DIS
LIN {X 98.364,Y 37.724,Z 67.000,A 180.000,B 0.000,C 180.000} C_DIS
LIN {X 97.969,Y 37.496,Z 67.000,A 180.000,B 0.000,C 180.000} C_DIS
LIN {X 97.790,Y 37.400,Z 67.000,A 180.000,B 0.000,C 180.000} C_DIS
LIN {X 97.361,Y 37.187,Z 67.000,A 180.000,B 0.000,C 180.000} C_DIS
LIN {X 97.254,Y 37.135,Z 67.000,A 180.000,B 0.000,C 180.000} C_DIS
LIN {X 97.075,Y 37.058,Z 67.000,A 180.000,B 0.000,C 180.000} C_DIS
LIN {X 96.718,Y 36.908,Z 67.000,A 180.000,B 0.000,C 180.000} C_DIS
LIN {X 96.539,Y 36.837,Z 67.000,A 180.000,B 0.000,C 180.000} C_DIS
LIN {X 96.520,Y 36.830,Z 67.000,A 180.000,B 0.000,C 180.000} C_DIS
LIN {X 96.360,Y 36.774,Z 67.000,A 180.000,B 0.000,C 180.000} C_DIS
LIN {X 96.003,Y 36.650,Z 67.000,A 180.000,B 0.000,C 180.000} C_DIS
LIN {X 95.824,Y 36.593,Z 67.000,A 180.000,B 0.000,C 180.000} C_DIS
LIN {X 95.288,Y 36.444,Z 67.000,A 180.000,B 0.000,C 180.000} C_DIS
LIN {X 95.109,Y 36.401,Z 67.000,A 180.000,B 0.000,C 180.000} C_DIS
LIN {X 94.601,Y 36.294,Z 67.000,A 180.000,B 0.000,C 180.000} C_DIS
LIN {X 94.573,Y 36.288,Z 67.000,A 180.000,B 0.000,C 180.000} C_DIS
LIN {X 94.394,Y 36.257,Z 67.000,A 180.000,B 0.000,C 180.000} C_DIS
LIN {X 94.036,Y 36.205,Z 67.000,A 180.000,B 0.000,C 180.000} C_DIS
LIN {X 93.857,Y 36.179,Z 67.000,A 180.000,B 0.000,C 180.000} C_DIS
LIN {X 93.679,Y 36.160,Z 67.000,A 180.000,B 0.000,C 180.000} C_DIS
LIN {X 93.321,Y 36.130,Z 67.000,A 180.000,B 0.000,C 180.000} C_DIS
LIN {X 93.142,Y 36.116,Z 67.000,A 180.000,B 0.000,C 180.000} C_DIS
LIN {X 93.130,Y 36.115,Z 67.000,A 180.000,B 0.000,C 180.000} C_DIS
LIN {X 92.964,Y 36.108,Z 67.000,A 180.000,B 0.000,C 180.000} C_DIS
LIN {X 92.606,Y 36.101,Z 67.000,A 180.000,B 0.000,C 180.000} C_DIS
LIN {X 92.427,Y 36.098,Z 67.000,A 180.000,B 0.000,C 180.000} C_DIS
LIN {X 92.249,Y 36.102,Z 67.000,A 180.000,B 0.000,C 180.000} C_DIS
LIN {X 91.891,Y 36.117,Z 67.000,A 180.000,B 0.000,C 180.000} C_DIS
LIN {X 91.712,Y 36.125,Z 67.000,A 180.000,B 0.000,C 180.000} C_DIS
LIN {X 91.533,Y 36.140,Z 67.000,A 180.000,B 0.000,C 180.000} C_DIS
LIN {X 91.019,Y 36.194,Z 67.000,A 180.000,B 0.000,C 180.000} C_DIS
LIN {X 91.008,Y 36.196,Z 67.000,A 180.000,B 0.000,C 180.000} C_DIS
LIN {X 91.007,Y 36.195,Z 67.000,A 180.000,B 0.000,C 180.000} C_DIS
LIN {X 91.003,Y 36.191,Z 67.000,A 180.000,B 0.000,C 180.000} C_DIS
LIN {X 90.997,Y 36.186,Z 67.000,A 180.000,B 0.000,C 180.000} C_DIS
LIN {X 90.917,Y 36.115,Z 67.000,A 180.000,B 0.000,C 180.000} C_DIS
LIN {X 90.818,Y 36.036,Z 67.000,A 180.000,B 0.000,C 180.000} C_DIS
LIN {X 90.677,Y 35.936,Z 67.000,A 180.000,B 0.000,C 180.000} C_DIS
LIN {X 90.640,Y 35.912,Z 67.000,A 180.000,B 0.000,C 180.000} C_DIS
LIN {X 90.461,Y 35.809,Z 67.000,A 180.000,B 0.000,C 180.000} C_DIS
LIN {X 90.356,Y 35.757,Z 67.000,A 180.000,B 0.000,C 180.000} C_DIS
LIN {X 90.282,Y 35.724,Z 67.000,A 180.000,B 0.000,C 180.000} C_DIS
LIN {X 90.103,Y 35.656,Z 67.000,A 180.000,B 0.000,C 180.000} C_DIS
LIN {X 89.925,Y 35.603,Z 67.000,A 180.000,B 0.000,C 180.000} C_DIS
LIN {X 89.819,Y 35.578,Z 67.000,A 180.000,B 0.000,C 180.000} C_DIS
LIN {X 89.746,Y 35.564,Z 67.000,A 180.000,B 0.000,C 180.000} C_DIS
LIN {X 89.567,Y 35.539,Z 67.000,A 180.000,B 0.000,C 180.000} C_DIS
LIN {X 89.388,Y 35.526,Z 67.000,A 180.000,B 0.000,C 180.000} C_DIS
LIN {X 89.209,Y 35.526,Z 67.000,A 180.000,B 0.000,C 180.000} C_DIS
LIN {X 89.031,Y 35.540,Z 67.000,A 180.000,B 0.000,C 180.000} C_DIS
LIN {X 88.852,Y 35.566,Z 67.000,A 180.000,B 0.000,C 180.000} C_DIS
LIN {X 88.788,Y 35.578,Z 67.000,A 180.000,B 0.000,C 180.000} C_DIS
LIN {X 88.673,Y 35.605,Z 67.000,A 180.000,B 0.000,C 180.000} C_DIS
LIN {X 88.494,Y 35.659,Z 67.000,A 180.000,B 0.000,C 180.000} C_DIS
LIN {X 45.590,Y 50.133,Z 67.000,A 180.000,B 0.000,C 180.000} C_DIS
LIN {X 45.411,Y 50.194,Z 67.000,A 180.000,B 0.000,C 180.000} C_DIS
LIN {X 45.296,Y 50.238,Z 67.000,A 180.000,B 0.000,C 180.000} C_DIS
LIN {X 45.232,Y 50.265,Z 67.000,A 180.000,B 0.000,C 180.000} C_DIS
LIN {X 45.053,Y 50.353,Z 67.000,A 180.000,B 0.000,C 180.000} C_DIS
LIN {X 44.944,Y 50.416,Z 67.000,A 180.000,B 0.000,C 180.000} C_DIS
LIN {X 44.874,Y 50.461,Z 67.000,A 180.000,B 0.000,C 180.000} C_DIS
LIN {X 44.785,Y 50.522,Z 67.000,A 180.000,B 0.000,C 180.000} C_DIS
LIN {X 44.696,Y 50.590,Z 67.000,A 180.000,B 0.000,C 180.000} C_DIS
LIN {X 44.689,Y 50.595,Z 67.000,A 180.000,B 0.000,C 180.000} C_DIS
LIN {X 44.603,Y 50.667,Z 67.000,A 180.000,B 0.000,C 180.000} C_DIS
LIN {X 44.517,Y 50.746,Z 67.000,A 180.000,B 0.000,C 180.000} C_DIS
LIN {X 44.488,Y 50.774,Z 67.000,A 180.000,B 0.000,C 180.000} C_DIS
LIN {X 44.410,Y 50.855,Z 67.000,A 180.000,B 0.000,C 180.000} C_DIS
LIN {X 44.338,Y 50.936,Z 67.000,A 180.000,B 0.000,C 180.000} C_DIS
LIN {X 44.325,Y 50.953,Z 67.000,A 180.000,B 0.000,C 180.000} C_DIS
LIN {X 44.254,Y 51.042,Z 67.000,A 180.000,B 0.000,C 180.000} C_DIS
LIN {X 44.189,Y 51.131,Z 67.000,A 180.000,B 0.000,C 180.000} C_DIS
LIN {X 44.159,Y 51.176,Z 67.000,A 180.000,B 0.000,C 180.000} C_DIS
LIN {X 44.077,Y 51.310,Z 67.000,A 180.000,B 0.000,C 180.000} C_DIS
LIN {X 43.984,Y 51.489,Z 67.000,A 180.000,B 0.000,C 180.000} C_DIS
LIN {X 43.981,Y 51.497,Z 67.000,A 180.000,B 0.000,C 180.000} C_DIS
LIN {X 43.909,Y 51.668,Z 67.000,A 180.000,B 0.000,C 180.000} C_DIS
LIN {X 43.849,Y 51.847,Z 67.000,A 180.000,B 0.000,C 180.000} C_DIS
LIN {X 43.804,Y 52.025,Z 67.000,A 180.000,B 0.000,C 180.000} C_DIS
LIN {X 43.802,Y 52.035,Z 67.000,A 180.000,B 0.000,C 180.000} C_DIS
LIN {X 43.772,Y 52.204,Z 67.000,A 180.000,B 0.000,C 180.000} C_DIS
LIN {X 43.754,Y 52.383,Z 67.000,A 180.000,B 0.000,C 180.000} C_DIS
LIN {X 43.748,Y 52.562,Z 67.000,A 180.000,B 0.000,C 180.000} C_DIS
LIN {X 43.756,Y 52.740,Z 67.000,A 180.000,B 0.000,C 180.000} C_DIS
LIN {X 43.776,Y 52.919,Z 67.000,A 180.000,B 0.000,C 180.000} C_DIS
LIN {X 43.802,Y 53.064,Z 67.000,A 180.000,B 0.000,C 180.000} C_DIS
LIN {X 43.809,Y 53.098,Z 67.000,A 180.000,B 0.000,C 180.000} C_DIS
LIN {X 43.856,Y 53.277,Z 67.000,A 180.000,B 0.000,C 180.000} C_DIS
LIN {X 43.916,Y 53.455,Z 67.000,A 180.000,B 0.000,C 180.000} C_DIS
LIN {X 50.248,Y 72.226,Z 67.000,A 180.000,B 0.000,C 180.000} C_DIS
LIN {X 50.311,Y 72.405,Z 67.000,A 180.000,B 0.000,C 180.000} C_DIS
LIN {X 50.388,Y 72.584,Z 67.000,A 180.000,B 0.000,C 180.000} C_DIS
LIN {X 50.416,Y 72.640,Z 67.000,A 180.000,B 0.000,C 180.000} C_DIS
LIN {X 50.484,Y 72.763,Z 67.000,A 180.000,B 0.000,C 180.000} C_DIS
LIN {X 50.595,Y 72.936,Z 67.000,A 180.000,B 0.000,C 180.000} C_DIS
LIN {X 50.599,Y 72.941,Z 67.000,A 180.000,B 0.000,C 180.000} C_DIS
LIN {X 50.665,Y 73.031,Z 67.000,A 180.000,B 0.000,C 180.000} C_DIS
LIN {X 50.737,Y 73.120,Z 67.000,A 180.000,B 0.000,C 180.000} C_DIS
LIN {X 50.774,Y 73.162,Z 67.000,A 180.000,B 0.000,C 180.000} C_DIS
LIN {X 50.905,Y 73.299,Z 67.000,A 180.000,B 0.000,C 180.000} C_DIS
LIN {X 50.953,Y 73.343,Z 67.000,A 180.000,B 0.000,C 180.000} C_DIS
LIN {X 51.112,Y 73.478,Z 67.000,A 180.000,B 0.000,C 180.000} C_DIS
LIN {X 51.131,Y 73.493,Z 67.000,A 180.000,B 0.000,C 180.000} C_DIS
LIN {X 51.310,Y 73.616,Z 67.000,A 180.000,B 0.000,C 180.000} C_DIS
LIN {X 51.376,Y 73.656,Z 67.000,A 180.000,B 0.000,C 180.000} C_DIS
LIN {X 51.489,Y 73.719,Z 67.000,A 180.000,B 0.000,C 180.000} C_DIS
LIN {X 51.668,Y 73.803,Z 67.000,A 180.000,B 0.000,C 180.000} C_DIS
LIN {X 51.749,Y 73.835,Z 67.000,A 180.000,B 0.000,C 180.000} C_DIS
LIN {X 51.847,Y 73.870,Z 67.000,A 180.000,B 0.000,C 180.000} C_DIS
LIN {X 52.025,Y 73.923,Z 67.000,A 180.000,B 0.000,C 180.000} C_DIS
LIN {X 52.204,Y 73.961,Z 67.000,A 180.000,B 0.000,C 180.000} C_DIS
LIN {X 52.383,Y 73.987,Z 67.000,A 180.000,B 0.000,C 180.000} C_DIS
LIN {X 52.562,Y 73.999,Z 67.000,A 180.000,B 0.000,C 180.000} C_DIS
LIN {X 52.740,Y 73.998,Z 67.000,A 180.000,B 0.000,C 180.000} C_DIS
LIN {X 52.919,Y 73.985,Z 67.000,A 180.000,B 0.000,C 180.000} C_DIS
LIN {X 53.098,Y 73.958,Z 67.000,A 180.000,B 0.000,C 180.000} C_DIS
LIN {X 53.277,Y 73.918,Z 67.000,A 180.000,B 0.000,C 180.000} C_DIS
LIN {X 53.455,Y 73.864,Z 67.000,A 180.000,B 0.000,C 180.000} C_DIS
LIN {X 76.321,Y 66.150,Z 67.000,A 180.000,B 0.000,C 180.000} C_DIS
LIN {X 96.464,Y 59.355,Z 67.000,A 180.000,B 0.000,C 180.000} C_DIS
LIN {X 96.539,Y 59.329,Z 67.000,A 180.000,B 0.000,C 180.000} C_DIS
LIN {X 96.718,Y 59.257,Z 67.000,A 180.000,B 0.000,C 180.000} C_DIS
LIN {X 96.883,Y 59.176,Z 67.000,A 180.000,B 0.000,C 180.000} C_DIS
LIN {X 96.897,Y 59.169,Z 67.000,A 180.000,B 0.000,C 180.000} C_DIS
LIN {X 97.075,Y 59.061,Z 67.000,A 180.000,B 0.000,C 180.000} C_DIS
LIN {X 97.167,Y 58.997,Z 67.000,A 180.000,B 0.000,C 180.000} C_DIS
LIN {X 97.254,Y 58.931,Z 67.000,A 180.000,B 0.000,C 180.000} C_DIS
LIN {X 97.385,Y 58.819,Z 67.000,A 180.000,B 0.000,C 180.000} C_DIS
LIN {X 97.433,Y 58.774,Z 67.000,A 180.000,B 0.000,C 180.000} C_DIS
LIN {X 97.562,Y 58.640,Z 67.000,A 180.000,B 0.000,C 180.000} C_DIS
LIN {X 97.612,Y 58.582,Z 67.000,A 180.000,B 0.000,C 180.000} C_DIS
LIN {X 97.707,Y 58.461,Z 67.000,A 180.000,B 0.000,C 180.000} C_DIS
LIN {X 97.790,Y 58.341,Z 67.000,A 180.000,B 0.000,C 180.000} C_DIS
LIN {X 97.828,Y 58.282,Z 67.000,A 180.000,B 0.000,C 180.000} C_DIS
LIN {X 97.928,Y 58.103,Z 67.000,A 180.000,B 0.000,C 180.000} C_DIS
LIN {X 97.969,Y 58.017,Z 67.000,A 180.000,B 0.000,C 180.000} C_DIS
LIN {X 98.009,Y 57.925,Z 67.000,A 180.000,B 0.000,C 180.000} C_DIS
LIN {X 98.075,Y 57.746,Z 67.000,A 180.000,B 0.000,C 180.000} C_DIS
LIN {X 98.125,Y 57.567,Z 67.000,A 180.000,B 0.000,C 180.000} C_DIS
LIN {X 98.148,Y 57.466,Z 67.000,A 180.000,B 0.000,C 180.000} C_DIS
LIN {X 98.155,Y 57.427,Z 67.000,A 180.000,B 0.000,C 180.000} C_DIS
LIN {X 98.159,Y 57.408,Z 67.000,A 180.000,B 0.000,C 180.000} C_DIS
LIN {X 98.161,Y 57.398,Z 67.000,A 180.000,B 0.000,C 180.000} C_DIS
LIN {X 98.177,Y 57.388,Z 67.000,A 180.000,B 0.000,C 180.000} C_DIS
LIN {X 98.505,Y 57.189,Z 67.000,A 180.000,B 0.000,C 180.000} C_DIS
LIN {X 98.684,Y 57.080,Z 67.000,A 180.000,B 0.000,C 180.000} C_DIS
LIN {X 98.760,Y 57.031,Z 67.000,A 180.000,B 0.000,C 180.000} C_DIS
LIN {X 98.863,Y 56.959,Z 67.000,A 180.000,B 0.000,C 180.000} C_DIS
LIN {X 99.221,Y 56.710,Z 67.000,A 180.000,B 0.000,C 180.000} C_DIS
LIN {X 99.273,Y 56.673,Z 67.000,A 180.000,B 0.000,C 180.000} C_DIS
LIN {X 99.399,Y 56.577,Z 67.000,A 180.000,B 0.000,C 180.000} C_DIS
LIN {X 99.757,Y 56.293,Z 67.000,A 180.000,B 0.000,C 180.000} C_DIS
LIN {X 99.936,Y 56.143,Z 67.000,A 180.000,B 0.000,C 180.000} C_DIS
LIN {X 100.339,Y 55.779,Z 67.000,A 180.000,B 0.000,C 180.000} C_DIS
LIN {X 100.472,Y 55.651,Z 67.000,A 180.000,B 0.000,C 180.000} C_DIS
LIN {X 100.829,Y 55.285,Z 67.000,A 180.000,B 0.000,C 180.000} C_DIS
LIN {X 100.870,Y 55.243,Z 67.000,A 180.000,B 0.000,C 180.000} C_DIS
LIN {X 101.008,Y 55.088,Z 67.000,A 180.000,B 0.000,C 180.000} C_DIS
LIN {X 101.187,Y 54.880,Z 67.000,A 180.000,B 0.000,C 180.000} C_DIS
LIN {X 101.336,Y 54.707,Z 67.000,A 180.000,B 0.000,C 180.000} C_DIS
LIN {X 101.366,Y 54.671,Z 67.000,A 180.000,B 0.000,C 180.000} C_DIS
LIN {X 101.476,Y 54.528,Z 67.000,A 180.000,B 0.000,C 180.000} C_DIS
LIN {X 101.747,Y 54.171,Z 67.000,A 180.000,B 0.000,C 180.000} C_DIS
LIN {X 101.872,Y 53.992,Z 67.000,A 180.000,B 0.000,C 180.000} C_DIS
LIN {X 102.109,Y 53.634,Z 67.000,A 180.000,B 0.000,C 180.000} C_DIS
LIN {X 102.224,Y 53.455,Z 67.000,A 180.000,B 0.000,C 180.000} C_DIS
LIN {X 102.260,Y 53.393,Z 67.000,A 180.000,B 0.000,C 180.000} C_DIS
LIN {X 102.438,Y 53.083,Z 67.000,A 180.000,B 0.000,C 180.000} C_DIS
LIN {X 102.533,Y 52.919,Z 67.000,A 180.000,B 0.000,C 180.000} C_DIS
LIN {X 102.617,Y 52.755,Z 67.000,A 180.000,B 0.000,C 180.000} C_DIS
LIN {X 102.802,Y 52.383,Z 67.000,A 180.000,B 0.000,C 180.000} C_DIS
LIN {X 102.887,Y 52.204,Z 67.000,A 180.000,B 0.000,C 180.000} C_DIS
LIN {X 102.963,Y 52.025,Z 67.000,A 180.000,B 0.000,C 180.000} C_DIS
LIN {X 103.113,Y 51.668,Z 67.000,A 180.000,B 0.000,C 180.000} C_DIS
LIN {X 103.153,Y 51.566,Z 67.000,A 180.000,B 0.000,C 180.000} C_DIS
LIN {X 103.181,Y 51.489,Z 67.000,A 180.000,B 0.000,C 180.000} C_DIS
LIN {X 103.332,Y 51.054,Z 67.000,A 180.000,B 0.000,C 180.000} C_DIS
LIN {X 103.367,Y 50.953,Z 67.000,A 180.000,B 0.000,C 180.000} C_DIS
LIN {X 103.421,Y 50.774,Z 67.000,A 180.000,B 0.000,C 180.000} C_DIS
LIN {X 103.520,Y 50.416,Z 67.000,A 180.000,B 0.000,C 180.000} C_DIS
LIN {X 103.569,Y 50.238,Z 67.000,A 180.000,B 0.000,C 180.000} C_DIS
LIN {X 103.609,Y 50.059,Z 67.000,A 180.000,B 0.000,C 180.000} C_DIS
LIN {X 103.690,Y 49.680,Z 67.000,A 180.000,B 0.000,C 180.000} C_DIS
LIN {X 103.722,Y 49.523,Z 67.000,A 180.000,B 0.000,C 180.000} C_DIS
LIN {X 103.750,Y 49.344,Z 67.000,A 180.000,B 0.000,C 180.000} C_DIS
LIN {X 103.803,Y 48.986,Z 67.000,A 180.000,B 0.000,C 180.000} C_DIS
LIN {X 103.828,Y 48.807,Z 67.000,A 180.000,B 0.000,C 180.000} C_DIS
LIN {X 103.844,Y 48.629,Z 67.000,A 180.000,B 0.000,C 180.000} C_DIS
LIN {X 103.874,Y 48.271,Z 67.000,A 180.000,B 0.000,C 180.000} C_DIS
LIN {X 103.888,Y 48.092,Z 67.000,A 180.000,B 0.000,C 180.000} C_DIS
LIN {X 103.893,Y 47.914,Z 67.000,A 180.000,B 0.000,C 180.000} C_DIS
LIN {X 103.900,Y 47.556,Z 67.000,A 180.000,B 0.000,C 180.000} C_DIS
LIN {X 103.902,Y 47.377,Z 67.000,A 180.000,B 0.000,C 180.000} C_DIS
LIN {X 103.896,Y 47.198,Z 67.000,A 180.000,B 0.000,C 180.000} C_DIS
LIN {X 103.881,Y 46.841,Z 67.000,A 180.000,B 0.000,C 180.000} C_DIS
LIN {X 103.872,Y 46.662,Z 67.000,A 180.000,B 0.000,C 180.000} C_DIS
LIN {X 103.869,Y 46.618,Z 67.000,A 180.000,B 0.000,C 180.000} C_DIS
LIN {X 103.855,Y 46.483,Z 67.000,A 180.000,B 0.000,C 180.000} C_DIS
LIN {X 103.836,Y 46.305,Z 67.000,A 180.000,B 0.000,C 180.000} C_DIS
; Link Move Starts
LIN {X 103.803,Y 45.992,Z 67.000,A 180.000,B 0.000,C 180.000} C_DIS
LIN {X 103.757,Y 45.698,Z 66.998,A 180.000,B 0.000,C 180.000} C_DIS
LIN {X 103.706,Y 45.388,Z 66.996,A 180.000,B 0.000,C 180.000} C_DIS
LIN {X 103.649,Y 45.096,Z 66.993,A 180.000,B 0.000,C 180.000} C_DIS
LIN {X 103.579,Y 44.789,Z 66.989,A 180.000,B 0.000,C 180.000} C_DIS
LIN {X 103.510,Y 44.494,Z 66.984,A 180.000,B 0.000,C 180.000} C_DIS
LIN {X 103.466,Y 44.345,Z 66.982,A 180.000,B 0.000,C 180.000} C_DIS
LIN {X 103.423,Y 44.196,Z 66.979,A 180.000,B 0.000,C 180.000} C_DIS
LIN {X 103.380,Y 44.045,Z 66.976,A 180.000,B 0.000,C 180.000} C_DIS
LIN {X 103.336,Y 43.894,Z 66.972,A 180.000,B 0.000,C 180.000} C_DIS
LIN {X 103.288,Y 43.752,Z 66.969,A 180.000,B 0.000,C 180.000} C_DIS
LIN {X 103.238,Y 43.612,Z 66.966,A 180.000,B 0.000,C 180.000} C_DIS
LIN {X 103.186,Y 43.464,Z 66.962,A 180.000,B 0.000,C 180.000} C_DIS
LIN {X 103.133,Y 43.316,Z 66.958,A 180.000,B 0.000,C 180.000} C_DIS
LIN {X 103.082,Y 43.174,Z 66.954,A 180.000,B 0.000,C 180.000} C_DIS
LIN {X 103.024,Y 43.035,Z 66.950,A 180.000,B 0.000,C 180.000} C_DIS
LIN {X 102.962,Y 42.891,Z 66.946,A 180.000,B 0.000,C 180.000} C_DIS
LIN {X 102.901,Y 42.747,Z 66.941,A 180.000,B 0.000,C 180.000} C_DIS
LIN {X 102.842,Y 42.608,Z 66.937,A 180.000,B 0.000,C 180.000} C_DIS
LIN {X 102.781,Y 42.471,Z 66.932,A 180.000,B 0.000,C 180.000} C_DIS
LIN {X 102.711,Y 42.330,Z 66.927,A 180.000,B 0.000,C 180.000} C_DIS
LIN {X 102.676,Y 42.260,Z 66.925,A 180.000,B 0.000,C 180.000} C_DIS
LIN {X 102.641,Y 42.190,Z 66.922,A 180.000,B 0.000,C 180.000} C_DIS
LIN {X 102.607,Y 42.121,Z 66.920,A 180.000,B 0.000,C 180.000} C_DIS
LIN {X 102.573,Y 42.052,Z 66.917,A 180.000,B 0.000,C 180.000} C_DIS
LIN {X 102.539,Y 41.984,Z 66.915,A 180.000,B 0.000,C 180.000} C_DIS
LIN {X 102.504,Y 41.915,Z 66.912,A 180.000,B 0.000,C 180.000} C_DIS
LIN {X 102.468,Y 41.847,Z 66.910,A 180.000,B 0.000,C 180.000} C_DIS
LIN {X 102.430,Y 41.780,Z 66.907,A 180.000,B 0.000,C 180.000} C_DIS
LIN {X 102.392,Y 41.713,Z 66.904,A 180.000,B 0.000,C 180.000} C_DIS
LIN {X 102.353,Y 41.646,Z 66.902,A 180.000,B 0.000,C 180.000} C_DIS
LIN {X 102.314,Y 41.578,Z 66.899,A 180.000,B 0.000,C 180.000} C_DIS
LIN {X 102.275,Y 41.510,Z 66.896,A 180.000,B 0.000,C 180.000} C_DIS
LIN {X 102.236,Y 41.442,Z 66.893,A 180.000,B 0.000,C 180.000} C_DIS
LIN {X 102.196,Y 41.374,Z 66.891,A 180.000,B 0.000,C 180.000} C_DIS
LIN {X 102.158,Y 41.309,Z 66.888,A 180.000,B 0.000,C 180.000} C_DIS
LIN {X 102.120,Y 41.244,Z 66.885,A 180.000,B 0.000,C 180.000} C_DIS
LIN {X 102.079,Y 41.180,Z 66.883,A 180.000,B 0.000,C 180.000} C_DIS
LIN {X 102.037,Y 41.117,Z 66.880,A 180.000,B 0.000,C 180.000} C_DIS
LIN {X 101.993,Y 41.051,Z 66.877,A 180.000,B 0.000,C 180.000} C_DIS
LIN {X 101.950,Y 40.986,Z 66.875,A 180.000,B 0.000,C 180.000} C_DIS
LIN {X 101.906,Y 40.920,Z 66.872,A 180.000,B 0.000,C 180.000} C_DIS
LIN {X 101.863,Y 40.854,Z 66.869,A 180.000,B 0.000,C 180.000} C_DIS
LIN {X 101.820,Y 40.791,Z 66.866,A 180.000,B 0.000,C 180.000} C_DIS
LIN {X 101.778,Y 40.727,Z 66.864,A 180.000,B 0.000,C 180.000} C_DIS
LIN {X 101.735,Y 40.664,Z 66.861,A 180.000,B 0.000,C 180.000} C_DIS
LIN {X 101.691,Y 40.602,Z 66.858,A 180.000,B 0.000,C 180.000} C_DIS
LIN {X 101.644,Y 40.540,Z 66.856,A 180.000,B 0.000,C 180.000} C_DIS
LIN {X 101.597,Y 40.477,Z 66.853,A 180.000,B 0.000,C 180.000} C_DIS
LIN {X 101.549,Y 40.415,Z 66.850,A 180.000,B 0.000,C 180.000} C_DIS
LIN {X 101.502,Y 40.353,Z 66.847,A 180.000,B 0.000,C 180.000} C_DIS
LIN {X 101.408,Y 40.229,Z 66.842,A 180.000,B 0.000,C 180.000} C_DIS
LIN {X 101.362,Y 40.168,Z 66.839,A 180.000,B 0.000,C 180.000} C_DIS
LIN {X 101.315,Y 40.106,Z 66.837,A 180.000,B 0.000,C 180.000} C_DIS
LIN {X 101.266,Y 40.046,Z 66.834,A 180.000,B 0.000,C 180.000} C_DIS
LIN {X 101.216,Y 39.987,Z 66.831,A 180.000,B 0.000,C 180.000} C_DIS
LIN {X 101.064,Y 39.811,Z 66.823,A 180.000,B 0.000,C 180.000} C_DIS
LIN {X 100.961,Y 39.691,Z 66.818,A 180.000,B 0.000,C 180.000} C_DIS
LIN {X 100.910,Y 39.632,Z 66.815,A 180.000,B 0.000,C 180.000} C_DIS
LIN {X 100.860,Y 39.574,Z 66.812,A 180.000,B 0.000,C 180.000} C_DIS
LIN {X 100.809,Y 39.517,Z 66.810,A 180.000,B 0.000,C 180.000} C_DIS
LIN {X 100.757,Y 39.462,Z 66.807,A 180.000,B 0.000,C 180.000} C_DIS
LIN {X 100.704,Y 39.408,Z 66.804,A 180.000,B 0.000,C 180.000} C_DIS
LIN {X 100.594,Y 39.295,Z 66.799,A 180.000,B 0.000,C 180.000} C_DIS
LIN {X 100.375,Y 39.072,Z 66.788,A 180.000,B 0.000,C 180.000} C_DIS
LIN {X 100.321,Y 39.017,Z 66.785,A 180.000,B 0.000,C 180.000} C_DIS
LIN {X 100.265,Y 38.964,Z 66.782,A 180.000,B 0.000,C 180.000} C_DIS
LIN {X 100.207,Y 38.912,Z 66.780,A 180.000,B 0.000,C 180.000} C_DIS
LIN {X 99.858,Y 38.598,Z 66.763,A 180.000,B 0.000,C 180.000} C_DIS
LIN {X 99.800,Y 38.546,Z 66.761,A 180.000,B 0.000,C 180.000} C_DIS
LIN {X 99.741,Y 38.496,Z 66.758,A 180.000,B 0.000,C 180.000} C_DIS
LIN {X 99.681,Y 38.447,Z 66.755,A 180.000,B 0.000,C 180.000} C_DIS
LIN {X 99.499,Y 38.303,Z 66.747,A 180.000,B 0.000,C 180.000} C_DIS
LIN {X 99.438,Y 38.255,Z 66.744,A 180.000,B 0.000,C 180.000} C_DIS
LIN {X 99.254,Y 38.110,Z 66.736,A 180.000,B 0.000,C 180.000} C_DIS
LIN {X 99.193,Y 38.063,Z 66.733,A 180.000,B 0.000,C 180.000} C_DIS
LIN {X 99.130,Y 38.018,Z 66.731,A 180.000,B 0.000,C 180.000} C_DIS
LIN {X 98.936,Y 37.885,Z 66.723,A 180.000,B 0.000,C 180.000} C_DIS
LIN {X 98.680,Y 37.708,Z 66.712,A 180.000,B 0.000,C 180.000} C_DIS
LIN {X 98.616,Y 37.664,Z 66.709,A 180.000,B 0.000,C 180.000} C_DIS
LIN {X 98.551,Y 37.623,Z 66.706,A 180.000,B 0.000,C 180.000} C_DIS
LIN {X 98.483,Y 37.582,Z 66.704,A 180.000,B 0.000,C 180.000} C_DIS
LIN {X 98.348,Y 37.501,Z 66.698,A 180.000,B 0.000,C 180.000} C_DIS
LIN {X 98.281,Y 37.461,Z 66.695,A 180.000,B 0.000,C 180.000} C_DIS
LIN {X 98.146,Y 37.380,Z 66.690,A 180.000,B 0.000,C 180.000} C_DIS
LIN {X 98.079,Y 37.339,Z 66.687,A 180.000,B 0.000,C 180.000} C_DIS
LIN {X 98.012,Y 37.299,Z 66.684,A 180.000,B 0.000,C 180.000} C_DIS
LIN {X 97.944,Y 37.261,Z 66.682,A 180.000,B 0.000,C 180.000} C_DIS
LIN {X 97.875,Y 37.225,Z 66.679,A 180.000,B 0.000,C 180.000} C_DIS
LIN {X 97.668,Y 37.117,Z 66.671,A 180.000,B 0.000,C 180.000} C_DIS
LIN {X 97.528,Y 37.045,Z 66.665,A 180.000,B 0.000,C 180.000} C_DIS
LIN {X 97.458,Y 37.008,Z 66.662,A 180.000,B 0.000,C 180.000} C_DIS
LIN {X 97.389,Y 36.973,Z 66.660,A 180.000,B 0.000,C 180.000} C_DIS
LIN {X 97.320,Y 36.938,Z 66.657,A 180.000,B 0.000,C 180.000} C_DIS
LIN {X 97.249,Y 36.906,Z 66.654,A 180.000,B 0.000,C 180.000} C_DIS
LIN {X 97.179,Y 36.875,Z 66.652,A 180.000,B 0.000,C 180.000} C_DIS
LIN {X 97.034,Y 36.811,Z 66.646,A 180.000,B 0.000,C 180.000} C_DIS
LIN {X 96.962,Y 36.779,Z 66.643,A 180.000,B 0.000,C 180.000} C_DIS
LIN {X 96.890,Y 36.748,Z 66.641,A 180.000,B 0.000,C 180.000} C_DIS
LIN {X 96.819,Y 36.716,Z 66.638,A 180.000,B 0.000,C 180.000} C_DIS
LIN {X 96.748,Y 36.685,Z 66.635,A 180.000,B 0.000,C 180.000} C_DIS
LIN {X 96.676,Y 36.654,Z 66.632,A 180.000,B 0.000,C 180.000} C_DIS
LIN {X 96.604,Y 36.625,Z 66.630,A 180.000,B 0.000,C 180.000} C_DIS
LIN {X 96.530,Y 36.598,Z 66.627,A 180.000,B 0.000,C 180.000} C_DIS
LIN {X 96.456,Y 36.571,Z 66.624,A 180.000,B 0.000,C 180.000} C_DIS
LIN {X 96.383,Y 36.544,Z 66.622,A 180.000,B 0.000,C 180.000} C_DIS
LIN {X 96.309,Y 36.516,Z 66.619,A 180.000,B 0.000,C 180.000} C_DIS
LIN {X 96.235,Y 36.489,Z 66.616,A 180.000,B 0.000,C 180.000} C_DIS
LIN {X 96.161,Y 36.462,Z 66.613,A 180.000,B 0.000,C 180.000} C_DIS
LIN {X 96.087,Y 36.435,Z 66.611,A 180.000,B 0.000,C 180.000} C_DIS
LIN {X 96.013,Y 36.408,Z 66.608,A 180.000,B 0.000,C 180.000} C_DIS
LIN {X 95.939,Y 36.383,Z 66.605,A 180.000,B 0.000,C 180.000} C_DIS
LIN {X 95.865,Y 36.360,Z 66.602,A 180.000,B 0.000,C 180.000} C_DIS
LIN {X 95.790,Y 36.338,Z 66.600,A 180.000,B 0.000,C 180.000} C_DIS
LIN {X 95.715,Y 36.316,Z 66.597,A 180.000,B 0.000,C 180.000} C_DIS
LIN {X 95.640,Y 36.293,Z 66.594,A 180.000,B 0.000,C 180.000} C_DIS
LIN {X 95.565,Y 36.271,Z 66.591,A 180.000,B 0.000,C 180.000} C_DIS
LIN {X 95.489,Y 36.248,Z 66.589,A 180.000,B 0.000,C 180.000} C_DIS
LIN {X 95.414,Y 36.226,Z 66.586,A 180.000,B 0.000,C 180.000} C_DIS
LIN {X 95.339,Y 36.204,Z 66.584,A 180.000,B 0.000,C 180.000} C_DIS
LIN {X 95.263,Y 36.183,Z 66.581,A 180.000,B 0.000,C 180.000} C_DIS
LIN {X 95.187,Y 36.164,Z 66.578,A 180.000,B 0.000,C 180.000} C_DIS
LIN {X 95.111,Y 36.147,Z 66.576,A 180.000,B 0.000,C 180.000} C_DIS
LIN {X 94.958,Y 36.112,Z 66.571,A 180.000,B 0.000,C 180.000} C_DIS
LIN {X 94.804,Y 36.076,Z 66.566,A 180.000,B 0.000,C 180.000} C_DIS
LIN {X 94.651,Y 36.042,Z 66.561,A 180.000,B 0.000,C 180.000} C_DIS
LIN {X 94.498,Y 36.010,Z 66.557,A 180.000,B 0.000,C 180.000} C_DIS
LIN {X 94.342,Y 35.985,Z 66.552,A 180.000,B 0.000,C 180.000} C_DIS
LIN {X 94.187,Y 35.960,Z 66.548,A 180.000,B 0.000,C 180.000} C_DIS
LIN {X 94.031,Y 35.935,Z 66.544,A 180.000,B 0.000,C 180.000} C_DIS
LIN {X 93.876,Y 35.910,Z 66.540,A 180.000,B 0.000,C 180.000} C_DIS
LIN {X 93.720,Y 35.892,Z 66.536,A 180.000,B 0.000,C 180.000} C_DIS
LIN {X 93.564,Y 35.877,Z 66.533,A 180.000,B 0.000,C 180.000} C_DIS
LIN {X 93.407,Y 35.862,Z 66.529,A 180.000,B 0.000,C 180.000} C_DIS
LIN {X 93.250,Y 35.848,Z 66.526,A 180.000,B 0.000,C 180.000} C_DIS
LIN {X 93.093,Y 35.835,Z 66.523,A 180.000,B 0.000,C 180.000} C_DIS
LIN {X 92.936,Y 35.829,Z 66.520,A 180.000,B 0.000,C 180.000} C_DIS
LIN {X 92.779,Y 35.824,Z 66.517,A 180.000,B 0.000,C 180.000} C_DIS
LIN {X 92.621,Y 35.820,Z 66.514,A 180.000,B 0.000,C 180.000} C_DIS
LIN {X 92.307,Y 35.815,Z 66.510,A 180.000,B 0.000,C 180.000} C_DIS
LIN {X 91.992,Y 35.826,Z 66.506,A 180.000,B 0.000,C 180.000} C_DIS
LIN {X 91.677,Y 35.838,Z 66.503,A 180.000,B 0.000,C 180.000} C_DIS
LIN {X 91.363,Y 35.868,Z 66.501,A 180.000,B 0.000,C 180.000} C_DIS
LIN {X 91.050,Y 35.900,Z 66.500,A 180.000,B 0.000,C 180.000} C_DIS
LIN {X 90.872,Y 35.926,Z 66.500,A 180.000,B 0.000,C 180.000} C_DIS
; Cutting Move Starts
LIN {X 90.818,Y 35.933,Z 66.500,A 180.000,B 0.000,C 180.000} C_DIS
LIN {X 90.702,Y 35.953,Z 66.500,A 180.000,B 0.000,C 180.000} C_DIS
LIN {X 90.693,Y 35.946,Z 66.500,A 180.000,B 0.000,C 180.000} C_DIS
LIN {X 90.677,Y 35.936,Z 66.500,A 180.000,B 0.000,C 180.000} C_DIS
LIN {X 90.640,Y 35.912,Z 66.500,A 180.000,B 0.000,C 180.000} C_DIS
LIN {X 90.461,Y 35.809,Z 66.500,A 180.000,B 0.000,C 180.000} C_DIS
LIN {X 90.356,Y 35.757,Z 66.500,A 180.000,B 0.000,C 180.000} C_DIS
LIN {X 90.282,Y 35.724,Z 66.500,A 180.000,B 0.000,C 180.000} C_DIS
LIN {X 90.103,Y 35.656,Z 66.500,A 180.000,B 0.000,C 180.000} C_DIS
LIN {X 89.925,Y 35.603,Z 66.500,A 180.000,B 0.000,C 180.000} C_DIS
LIN {X 89.819,Y 35.578,Z 66.500,A 180.000,B 0.000,C 180.000} C_DIS
LIN {X 89.746,Y 35.564,Z 66.500,A 180.000,B 0.000,C 180.000} C_DIS
LIN {X 89.567,Y 35.539,Z 66.500,A 180.000,B 0.000,C 180.000} C_DIS
LIN {X 89.388,Y 35.526,Z 66.500,A 180.000,B 0.000,C 180.000} C_DIS
LIN {X 89.209,Y 35.526,Z 66.500,A 180.000,B 0.000,C 180.000} C_DIS
LIN {X 89.031,Y 35.540,Z 66.500,A 180.000,B 0.000,C 180.000} C_DIS
LIN {X 88.852,Y 35.566,Z 66.500,A 180.000,B 0.000,C 180.000} C_DIS
LIN {X 88.788,Y 35.578,Z 66.500,A 180.000,B 0.000,C 180.000} C_DIS
LIN {X 88.673,Y 35.605,Z 66.500,A 180.000,B 0.000,C 180.000} C_DIS
LIN {X 88.494,Y 35.659,Z 66.500,A 180.000,B 0.000,C 180.000} C_DIS
LIN {X 45.590,Y 50.133,Z 66.500,A 180.000,B 0.000,C 180.000} C_DIS
LIN {X 45.411,Y 50.194,Z 66.500,A 180.000,B 0.000,C 180.000} C_DIS
LIN {X 45.296,Y 50.238,Z 66.500,A 180.000,B 0.000,C 180.000} C_DIS
LIN {X 45.232,Y 50.265,Z 66.500,A 180.000,B 0.000,C 180.000} C_DIS
LIN {X 45.053,Y 50.353,Z 66.500,A 180.000,B 0.000,C 180.000} C_DIS
LIN {X 44.944,Y 50.416,Z 66.500,A 180.000,B 0.000,C 180.000} C_DIS
LIN {X 44.874,Y 50.461,Z 66.500,A 180.000,B 0.000,C 180.000} C_DIS
LIN {X 44.785,Y 50.522,Z 66.500,A 180.000,B 0.000,C 180.000} C_DIS
LIN {X 44.696,Y 50.590,Z 66.500,A 180.000,B 0.000,C 180.000} C_DIS
LIN {X 44.689,Y 50.595,Z 66.500,A 180.000,B 0.000,C 180.000} C_DIS
LIN {X 44.603,Y 50.667,Z 66.500,A 180.000,B 0.000,C 180.000} C_DIS
LIN {X 44.517,Y 50.746,Z 66.500,A 180.000,B 0.000,C 180.000} C_DIS
LIN {X 44.488,Y 50.774,Z 66.500,A 180.000,B 0.000,C 180.000} C_DIS
LIN {X 44.410,Y 50.855,Z 66.500,A 180.000,B 0.000,C 180.000} C_DIS
LIN {X 44.338,Y 50.936,Z 66.500,A 180.000,B 0.000,C 180.000} C_DIS
LIN {X 44.325,Y 50.953,Z 66.500,A 180.000,B 0.000,C 180.000} C_DIS
LIN {X 44.254,Y 51.042,Z 66.500,A 180.000,B 0.000,C 180.000} C_DIS
LIN {X 44.189,Y 51.131,Z 66.500,A 180.000,B 0.000,C 180.000} C_DIS
LIN {X 44.159,Y 51.176,Z 66.500,A 180.000,B 0.000,C 180.000} C_DIS
LIN {X 44.077,Y 51.310,Z 66.500,A 180.000,B 0.000,C 180.000} C_DIS
LIN {X 43.984,Y 51.489,Z 66.500,A 180.000,B 0.000,C 180.000} C_DIS
LIN {X 43.981,Y 51.497,Z 66.500,A 180.000,B 0.000,C 180.000} C_DIS
LIN {X 43.909,Y 51.668,Z 66.500,A 180.000,B 0.000,C 180.000} C_DIS
LIN {X 43.849,Y 51.847,Z 66.500,A 180.000,B 0.000,C 180.000} C_DIS
LIN {X 43.804,Y 52.025,Z 66.500,A 180.000,B 0.000,C 180.000} C_DIS
LIN {X 43.802,Y 52.035,Z 66.500,A 180.000,B 0.000,C 180.000} C_DIS
LIN {X 43.772,Y 52.204,Z 66.500,A 180.000,B 0.000,C 180.000} C_DIS
LIN {X 43.754,Y 52.383,Z 66.500,A 180.000,B 0.000,C 180.000} C_DIS
LIN {X 43.748,Y 52.562,Z 66.500,A 180.000,B 0.000,C 180.000} C_DIS
LIN {X 43.756,Y 52.740,Z 66.500,A 180.000,B 0.000,C 180.000} C_DIS
LIN {X 43.776,Y 52.919,Z 66.500,A 180.000,B 0.000,C 180.000} C_DIS
LIN {X 43.802,Y 53.064,Z 66.500,A 180.000,B 0.000,C 180.000} C_DIS
LIN {X 43.809,Y 53.098,Z 66.500,A 180.000,B 0.000,C 180.000} C_DIS
LIN {X 43.856,Y 53.277,Z 66.500,A 180.000,B 0.000,C 180.000} C_DIS
LIN {X 43.916,Y 53.455,Z 66.500,A 180.000,B 0.000,C 180.000} C_DIS
LIN {X 50.248,Y 72.226,Z 66.500,A 180.000,B 0.000,C 180.000} C_DIS
LIN {X 50.311,Y 72.405,Z 66.500,A 180.000,B 0.000,C 180.000} C_DIS
LIN {X 50.388,Y 72.584,Z 66.500,A 180.000,B 0.000,C 180.000} C_DIS
LIN {X 50.416,Y 72.640,Z 66.500,A 180.000,B 0.000,C 180.000} C_DIS
LIN {X 50.484,Y 72.763,Z 66.500,A 180.000,B 0.000,C 180.000} C_DIS
LIN {X 50.595,Y 72.936,Z 66.500,A 180.000,B 0.000,C 180.000} C_DIS
LIN {X 50.599,Y 72.941,Z 66.500,A 180.000,B 0.000,C 180.000} C_DIS
LIN {X 50.665,Y 73.031,Z 66.500,A 180.000,B 0.000,C 180.000} C_DIS
LIN {X 50.737,Y 73.120,Z 66.500,A 180.000,B 0.000,C 180.000} C_DIS
LIN {X 50.774,Y 73.162,Z 66.500,A 180.000,B 0.000,C 180.000} C_DIS
LIN {X 50.905,Y 73.299,Z 66.500,A 180.000,B 0.000,C 180.000} C_DIS
LIN {X 50.953,Y 73.343,Z 66.500,A 180.000,B 0.000,C 180.000} C_DIS
LIN {X 51.112,Y 73.478,Z 66.500,A 180.000,B 0.000,C 180.000} C_DIS
LIN {X 51.131,Y 73.493,Z 66.500,A 180.000,B 0.000,C 180.000} C_DIS
LIN {X 51.310,Y 73.616,Z 66.500,A 180.000,B 0.000,C 180.000} C_DIS
LIN {X 51.376,Y 73.656,Z 66.500,A 180.000,B 0.000,C 180.000} C_DIS
LIN {X 51.489,Y 73.719,Z 66.500,A 180.000,B 0.000,C 180.000} C_DIS
LIN {X 51.668,Y 73.803,Z 66.500,A 180.000,B 0.000,C 180.000} C_DIS
LIN {X 51.749,Y 73.835,Z 66.500,A 180.000,B 0.000,C 180.000} C_DIS
LIN {X 51.847,Y 73.870,Z 66.500,A 180.000,B 0.000,C 180.000} C_DIS
LIN {X 52.025,Y 73.923,Z 66.500,A 180.000,B 0.000,C 180.000} C_DIS
LIN {X 52.204,Y 73.961,Z 66.500,A 180.000,B 0.000,C 180.000} C_DIS
LIN {X 52.383,Y 73.987,Z 66.500,A 180.000,B 0.000,C 180.000} C_DIS
LIN {X 52.562,Y 73.999,Z 66.500,A 180.000,B 0.000,C 180.000} C_DIS
LIN {X 52.740,Y 73.998,Z 66.500,A 180.000,B 0.000,C 180.000} C_DIS
LIN {X 52.919,Y 73.985,Z 66.500,A 180.000,B 0.000,C 180.000} C_DIS
LIN {X 53.098,Y 73.958,Z 66.500,A 180.000,B 0.000,C 180.000} C_DIS
LIN {X 53.277,Y 73.918,Z 66.500,A 180.000,B 0.000,C 180.000} C_DIS
LIN {X 53.455,Y 73.864,Z 66.500,A 180.000,B 0.000,C 180.000} C_DIS
LIN {X 83.198,Y 63.830,Z 66.500,A 180.000,B 0.000,C 180.000} C_DIS
LIN {X 96.464,Y 59.355,Z 66.500,A 180.000,B 0.000,C 180.000} C_DIS
LIN {X 96.539,Y 59.329,Z 66.500,A 180.000,B 0.000,C 180.000} C_DIS
LIN {X 96.718,Y 59.257,Z 66.500,A 180.000,B 0.000,C 180.000} C_DIS
LIN {X 96.883,Y 59.176,Z 66.500,A 180.000,B 0.000,C 180.000} C_DIS
LIN {X 96.897,Y 59.169,Z 66.500,A 180.000,B 0.000,C 180.000} C_DIS
LIN {X 97.075,Y 59.061,Z 66.500,A 180.000,B 0.000,C 180.000} C_DIS
LIN {X 97.167,Y 58.997,Z 66.500,A 180.000,B 0.000,C 180.000} C_DIS
LIN {X 97.254,Y 58.931,Z 66.500,A 180.000,B 0.000,C 180.000} C_DIS
LIN {X 97.385,Y 58.819,Z 66.500,A 180.000,B 0.000,C 180.000} C_DIS
LIN {X 97.433,Y 58.774,Z 66.500,A 180.000,B 0.000,C 180.000} C_DIS
LIN {X 97.562,Y 58.640,Z 66.500,A 180.000,B 0.000,C 180.000} C_DIS
LIN {X 97.612,Y 58.582,Z 66.500,A 180.000,B 0.000,C 180.000} C_DIS
LIN {X 97.707,Y 58.461,Z 66.500,A 180.000,B 0.000,C 180.000} C_DIS
LIN {X 97.790,Y 58.341,Z 66.500,A 180.000,B 0.000,C 180.000} C_DIS
LIN {X 97.828,Y 58.282,Z 66.500,A 180.000,B 0.000,C 180.000} C_DIS
LIN {X 97.928,Y 58.103,Z 66.500,A 180.000,B 0.000,C 180.000} C_DIS
LIN {X 97.969,Y 58.017,Z 66.500,A 180.000,B 0.000,C 180.000} C_DIS
LIN {X 98.009,Y 57.925,Z 66.500,A 180.000,B 0.000,C 180.000} C_DIS
LIN {X 98.044,Y 57.835,Z 66.500,A 180.000,B 0.000,C 180.000} C_DIS
LIN {X 98.060,Y 57.791,Z 66.500,A 180.000,B 0.000,C 180.000} C_DIS
LIN {X 98.063,Y 57.781,Z 66.500,A 180.000,B 0.000,C 180.000} C_DIS
LIN {X 98.064,Y 57.777,Z 66.500,A 180.000,B 0.000,C 180.000} C_DIS
LIN {X 98.066,Y 57.776,Z 66.500,A 180.000,B 0.000,C 180.000} C_DIS
LIN {X 98.148,Y 57.733,Z 66.500,A 180.000,B 0.000,C 180.000} C_DIS
LIN {X 98.327,Y 57.633,Z 66.500,A 180.000,B 0.000,C 180.000} C_DIS
LIN {X 98.729,Y 57.388,Z 66.500,A 180.000,B 0.000,C 180.000} C_DIS
LIN {X 98.863,Y 57.306,Z 66.500,A 180.000,B 0.000,C 180.000} C_DIS
LIN {X 99.005,Y 57.210,Z 66.500,A 180.000,B 0.000,C 180.000} C_DIS
LIN {X 99.399,Y 56.935,Z 66.500,A 180.000,B 0.000,C 180.000} C_DIS
LIN {X 99.513,Y 56.852,Z 66.500,A 180.000,B 0.000,C 180.000} C_DIS
LIN {X 99.578,Y 56.801,Z 66.500,A 180.000,B 0.000,C 180.000} C_DIS
LIN {X 99.964,Y 56.495,Z 66.500,A 180.000,B 0.000,C 180.000} C_DIS
LIN {X 100.114,Y 56.368,Z 66.500,A 180.000,B 0.000,C 180.000} C_DIS
LIN {X 100.472,Y 56.046,Z 66.500,A 180.000,B 0.000,C 180.000} C_DIS
LIN {X 100.569,Y 55.958,Z 66.500,A 180.000,B 0.000,C 180.000} C_DIS
LIN {X 100.651,Y 55.878,Z 66.500,A 180.000,B 0.000,C 180.000} C_DIS
LIN {X 101.008,Y 55.513,Z 66.500,A 180.000,B 0.000,C 180.000} C_DIS
LIN {X 101.096,Y 55.422,Z 66.500,A 180.000,B 0.000,C 180.000} C_DIS
LIN {X 101.187,Y 55.320,Z 66.500,A 180.000,B 0.000,C 180.000} C_DIS
LIN {X 101.407,Y 55.064,Z 66.500,A 180.000,B 0.000,C 180.000} C_DIS
LIN {X 101.545,Y 54.905,Z 66.500,A 180.000,B 0.000,C 180.000} C_DIS
LIN {X 101.561,Y 54.886,Z 66.500,A 180.000,B 0.000,C 180.000} C_DIS
LIN {X 101.700,Y 54.707,Z 66.500,A 180.000,B 0.000,C 180.000} C_DIS
LIN {X 101.971,Y 54.349,Z 66.500,A 180.000,B 0.000,C 180.000} C_DIS
LIN {X 102.081,Y 54.196,Z 66.500,A 180.000,B 0.000,C 180.000} C_DIS
LIN {X 102.335,Y 53.813,Z 66.500,A 180.000,B 0.000,C 180.000} C_DIS
LIN {X 102.438,Y 53.655,Z 66.500,A 180.000,B 0.000,C 180.000} C_DIS
LIN {X 102.451,Y 53.634,Z 66.500,A 180.000,B 0.000,C 180.000} C_DIS
LIN {X 102.555,Y 53.455,Z 66.500,A 180.000,B 0.000,C 180.000} C_DIS
LIN {X 102.761,Y 53.098,Z 66.500,A 180.000,B 0.000,C 180.000} C_DIS
LIN {X 102.796,Y 53.036,Z 66.500,A 180.000,B 0.000,C 180.000} C_DIS
LIN {X 102.856,Y 52.919,Z 66.500,A 180.000,B 0.000,C 180.000} C_DIS
LIN {X 103.033,Y 52.562,Z 66.500,A 180.000,B 0.000,C 180.000} C_DIS
LIN {X 103.121,Y 52.383,Z 66.500,A 180.000,B 0.000,C 180.000} C_DIS
LIN {X 103.153,Y 52.311,Z 66.500,A 180.000,B 0.000,C 180.000} C_DIS
LIN {X 103.199,Y 52.204,Z 66.500,A 180.000,B 0.000,C 180.000} C_DIS
LIN {X 103.349,Y 51.847,Z 66.500,A 180.000,B 0.000,C 180.000} C_DIS
LIN {X 103.422,Y 51.668,Z 66.500,A 180.000,B 0.000,C 180.000} C_DIS
LIN {X 103.485,Y 51.489,Z 66.500,A 180.000,B 0.000,C 180.000} C_DIS
LIN {X 103.609,Y 51.131,Z 66.500,A 180.000,B 0.000,C 180.000} C_DIS
LIN {X 103.668,Y 50.953,Z 66.500,A 180.000,B 0.000,C 180.000} C_DIS
LIN {X 103.690,Y 50.876,Z 66.500,A 180.000,B 0.000,C 180.000} C_DIS
LIN {X 103.818,Y 50.416,Z 66.500,A 180.000,B 0.000,C 180.000} C_DIS
LIN {X 103.864,Y 50.238,Z 66.500,A 180.000,B 0.000,C 180.000} C_DIS
LIN {X 103.869,Y 50.219,Z 66.500,A 180.000,B 0.000,C 180.000} C_DIS
LIN {X 103.903,Y 50.059,Z 66.500,A 180.000,B 0.000,C 180.000} C_DIS
LIN {X 103.978,Y 49.701,Z 66.500,A 180.000,B 0.000,C 180.000} C_DIS
LIN {X 104.013,Y 49.523,Z 66.500,A 180.000,B 0.000,C 180.000} C_DIS
LIN {X 104.040,Y 49.344,Z 66.500,A 180.000,B 0.000,C 180.000} C_DIS
LIN {X 104.092,Y 48.986,Z 66.500,A 180.000,B 0.000,C 180.000} C_DIS
LIN {X 104.116,Y 48.807,Z 66.500,A 180.000,B 0.000,C 180.000} C_DIS
LIN {X 104.132,Y 48.629,Z 66.500,A 180.000,B 0.000,C 180.000} C_DIS
LIN {X 104.162,Y 48.271,Z 66.500,A 180.000,B 0.000,C 180.000} C_DIS
LIN {X 104.175,Y 48.092,Z 66.500,A 180.000,B 0.000,C 180.000} C_DIS
LIN {X 104.179,Y 47.914,Z 66.500,A 180.000,B 0.000,C 180.000} C_DIS
LIN {X 104.187,Y 47.556,Z 66.500,A 180.000,B 0.000,C 180.000} C_DIS
LIN {X 104.189,Y 47.377,Z 66.500,A 180.000,B 0.000,C 180.000} C_DIS
LIN {X 104.183,Y 47.198,Z 66.500,A 180.000,B 0.000,C 180.000} C_DIS
